LIN {X 0.029,Y -586.530,Z 530.477,A 0.000,B 0.000,C 90.000,E1 301.799} C_DIS
LIN {X 0.083,Y -590.989,Z 530.474,A 0.000,B 0.000,C 90.000,E1 301.258} C_DIS
LIN {X 0.018,Y -595.734,Z 530.471,A 0.000,B 0.000,C 90.000,E1 300.747} C_DIS
LIN {X 0.138,Y -599.927,Z 530.468,A 0.000,B 0.000,C 90.000,E1 300.207} C_DIS
LIN {X 0.251,Y -604.747,Z 530.464,A 0.000,B 0.000,C 90.000,E1 299.539} C_DIS
LIN {X 0.334,Y -611.596,Z 530.458,A 0.000,B 0.000,C 90.000,E1 298.487} C_DIS
LIN {X 0.265,Y -614.592,Z 530.456,A 0.000,B 0.000,C 90.000,E1 297.975} C_DIS
LIN {X 0.227,Y -616.501,Z 530.453,A 0.000,B 0.000,C 90.000,E1 297.590} C_DIS
LIN {X 0.209,Y -617.579,Z 530.452,A 0.000,B 0.000,C 90.000,E1 297.334} C_DIS
LIN {X 0.179,Y -619.100,Z 530.449,A 0.000,B 0.000,C 90.000,E1 296.821} C_DIS
LIN {X 0.170,Y -619.570,Z 530.448,A 0.000,B 0.000,C 90.000,E1 296.565} C_DIS
LIN {X 0.162,Y -619.896,Z 530.446,A 0.000,B 0.000,C 90.000,E1 296.309} C_DIS
LIN {X 0.157,Y -620.039,Z 530.445,A 0.000,B 0.000,C 90.000,E1 296.052} C_DIS
LIN {X 0.146,Y -619.660,Z 530.442,A 0.000,B 0.000,C 90.000,E1 295.540} C_DIS
LIN {X 0.140,Y -619.341,Z 530.441,A 0.000,B 0.000,C 90.000,E1 295.283} C_DIS
LIN {X 0.133,Y -618.398,Z 530.439,A 0.000,B 0.000,C 90.000,E1 295.027} C_DIS
LIN {X 0.123,Y -617.735,Z 530.438,A 0.000,B 0.000,C 90.000,E1 294.771} C_DIS
LIN {X 0.117,Y -617.127,Z 530.437,A 0.000,B 0.000,C 90.000,E1 294.643} C_DIS
LIN {X 0.110,Y -616.003,Z 530.436,A 0.000,B 0.000,C 90.000,E1 294.515} C_DIS
LIN {X 0.101,Y -615.099,Z 530.436,A 0.000,B 0.000,C 90.000,E1 294.387} C_DIS
LIN {X 0.079,Y -613.630,Z 530.434,A 0.000,B 0.000,C 90.000,E1 294.131} C_DIS
LIN {X -0.183,Y -612.297,Z 530.433,A 0.000,B 0.000,C 90.000,E1 294.027} C_DIS
LIN {X -0.142,Y -610.741,Z 530.433,A 0.000,B 0.000,C 90.000,E1 293.898} C_DIS
LIN {X -0.099,Y -607.183,Z 530.431,A 0.000,B 0.000,C 90.000,E1 293.567} C_DIS
LIN {X -0.081,Y -600.309,Z 530.429,A 0.000,B 0.000,C 90.000,E1 293.131} C_DIS
LIN {X 0.139,Y -594.236,Z 530.427,A 0.000,B 0.000,C 90.000,E1 292.845} C_DIS
LIN {X -0.178,Y -586.014,Z 530.425,A 0.000,B 0.000,C 90.000,E1 292.514} C_DIS
LIN {X 0.007,Y -580.558,Z 530.423,A 0.000,B 0.000,C 90.000,E1 292.206} C_DIS
LIN {X -0.138,Y -578.106,Z 530.422,A 0.000,B 0.000,C 90.000,E1 292.025} C_DIS
LIN {X -0.120,Y -576.577,Z 530.421,A 0.000,B 0.000,C 90.000,E1 291.844} C_DIS
LIN {X -0.128,Y -575.849,Z 530.420,A 0.000,B 0.000,C 90.000,E1 291.642} C_DIS
LIN {X 0.113,Y -575.619,Z 530.419,A 0.000,B 0.000,C 90.000,E1 291.461} C_DIS
LIN {X -0.080,Y -575.495,Z 530.414,A 0.000,B 0.000,C 90.000,E1 290.482} C_DIS
LIN {X 0.294,Y -575.816,Z 530.409,A 0.000,B 0.000,C 90.000,E1 289.631} C_DIS
LIN {X -0.234,Y -575.885,Z 530.403,A 0.000,B 0.000,C 90.000,E1 288.598} C_DIS
LIN {X -0.026,Y -575.856,Z 530.396,A 0.000,B 0.000,C 90.000,E1 287.221} C_DIS
LIN {X 0.184,Y -575.564,Z 530.388,A 0.000,B 0.000,C 90.000,E1 285.843} C_DIS
LIN {X 0.081,Y -574.849,Z 530.378,A 0.000,B 0.000,C 90.000,E1 283.953} C_DIS
LIN {X 0.114,Y -574.340,Z 530.370,A 0.000,B 0.000,C 90.000,E1 282.591} C_DIS
LIN {X 0.204,Y -573.645,Z 530.361,A 0.000,B 0.000,C 90.000,E1 280.950} C_DIS
LIN {X 0.169,Y -572.922,Z 530.352,A 0.000,B 0.000,C 90.000,E1 279.321} C_DIS
LIN {X -0.235,Y -572.026,Z 530.340,A 0.000,B 0.000,C 90.000,E1 277.182} C_DIS
LIN {X -0.193,Y -571.609,Z 530.334,A 0.000,B 0.000,C 90.000,E1 276.087} C_DIS
LIN {X 0.016,Y -571.061,Z 530.326,A 0.000,B 0.000,C 90.000,E1 274.702} C_DIS
LIN {X 0.120,Y -570.353,Z 530.319,A 0.000,B 0.000,C 90.000,E1 273.326} C_DIS
LIN {X 0.094,Y -569.713,Z 530.313,A 0.000,B 0.000,C 90.000,E1 272.236} C_DIS
LIN {X 0.179,Y -568.765,Z 530.305,A 0.000,B 0.000,C 90.000,E1 270.859} C_DIS
LIN {X 0.111,Y -567.916,Z 530.299,A 0.000,B 0.000,C 90.000,E1 269.771} C_DIS
LIN {X -0.167,Y -566.298,Z 530.288,A 0.000,B 0.000,C 90.000,E1 267.879} C_DIS
LIN {X -0.032,Y -564.887,Z 530.279,A 0.000,B 0.000,C 90.000,E1 266.216} C_DIS
LIN {X 0.000,Y -563.746,Z 530.271,A 0.000,B 0.000,C 90.000,E1 264.837} C_DIS
LIN {X 0.072,Y -562.379,Z 530.264,A 0.000,B 0.000,C 90.000,E1 263.451} C_DIS
LIN {X -0.024,Y -561.272,Z 530.258,A 0.000,B 0.000,C 90.000,E1 262.356} C_DIS
LIN {X -0.002,Y -559.763,Z 530.250,A 0.000,B 0.000,C 90.000,E1 260.971} C_DIS
LIN {X 0.212,Y -557.715,Z 530.241,A 0.000,B 0.000,C 90.000,E1 259.285} C_DIS
LIN {X -0.058,Y -555.607,Z 530.231,A 0.000,B 0.000,C 90.000,E1 257.645} C_DIS
LIN {X 0.046,Y -554.014,Z 530.225,A 0.000,B 0.000,C 90.000,E1 256.520} C_DIS
LIN {X 0.113,Y -551.877,Z 530.217,A 0.000,B 0.000,C 90.000,E1 255.117} C_DIS
LIN {X -0.117,Y -549.518,Z 530.210,A 0.000,B 0.000,C 90.000,E1 253.740} C_DIS
LIN {X -0.196,Y -548.025,Z 530.205,A 0.000,B 0.000,C 90.000,E1 252.906} C_DIS
LIN {X 0.199,Y -545.202,Z 530.197,A 0.000,B 0.000,C 90.000,E1 251.456} C_DIS
LIN {X -0.211,Y -542.867,Z 530.191,A 0.000,B 0.000,C 90.000,E1 250.369} C_DIS
LIN {X 0.039,Y -540.458,Z 530.185,A 0.000,B 0.000,C 90.000,E1 249.209} C_DIS
LIN {X -0.252,Y -537.864,Z 530.178,A 0.000,B 0.000,C 90.000,E1 248.103} C_DIS
LIN {X 0.119,Y -535.177,Z 530.172,A 0.000,B 0.000,C 90.000,E1 246.922} C_DIS
LIN {X -0.040,Y -532.319,Z 530.166,A 0.000,B 0.000,C 90.000,E1 245.793} C_DIS
LIN {X -0.240,Y -529.288,Z 530.159,A 0.000,B 0.000,C 90.000,E1 244.665} C_DIS
LIN {X -0.092,Y -525.356,Z 530.151,A 0.000,B 0.000,C 90.000,E1 243.204} C_DIS
LIN {X 0.140,Y -520.454,Z 530.141,A 0.000,B 0.000,C 90.000,E1 241.435} C_DIS
LIN {X -0.096,Y -516.317,Z 530.133,A 0.000,B 0.000,C 90.000,E1 239.999} C_DIS
LIN {X -0.157,Y -513.781,Z 530.128,A 0.000,B 0.000,C 90.000,E1 239.125} C_DIS
LIN {X 0.075,Y -508.474,Z 530.119,A 0.000,B 0.000,C 90.000,E1 237.327} C_DIS
LIN {X 0.100,Y -504.834,Z 530.112,A 0.000,B 0.000,C 90.000,E1 236.135} C_DIS
LIN {X 0.283,Y -496.859,Z 530.097,A 0.000,B 0.000,C 90.000,E1 233.417} C_DIS
LIN {X 0.143,Y -491.747,Z 530.087,A 0.000,B 0.000,C 90.000,E1 231.618} C_DIS
LIN {X -0.039,Y -485.884,Z 530.075,A 0.000,B 0.000,C 90.000,E1 229.504} C_DIS
LIN {X 0.314,Y -480.233,Z 530.063,A 0.000,B 0.000,C 90.000,E1 227.310} C_DIS
LIN {X 0.128,Y -474.745,Z 530.051,A 0.000,B 0.000,C 90.000,E1 225.162} C_DIS
LIN {X 0.041,Y -470.153,Z 530.041,A 0.000,B 0.000,C 90.000,E1 223.299} C_DIS
LIN {X -0.203,Y -466.470,Z 530.032,A 0.000,B 0.000,C 90.000,E1 221.757} C_DIS
LIN {X -0.162,Y -462.896,Z 530.023,A 0.000,B 0.000,C 90.000,E1 220.172} C_DIS
LIN {X -0.071,Y -457.922,Z 530.011,A 0.000,B 0.000,C 90.000,E1 217.935} C_DIS
LIN {X -0.044,Y -453.772,Z 530.000,A 0.000,B 0.000,C 90.000,E1 216.011} C_DIS
LIN {X -0.292,Y -449.120,Z 529.988,A 0.000,B 0.000,C 90.000,E1 213.785} C_DIS
LIN {X 0.017,Y -445.273,Z 529.977,A 0.000,B 0.000,C 90.000,E1 211.799} C_DIS
LIN {X -0.233,Y -441.608,Z 529.966,A 0.000,B 0.000,C 90.000,E1 209.873} C_DIS
LIN {X 0.062,Y -436.926,Z 529.951,A 0.000,B 0.000,C 90.000,E1 207.206} C_DIS
LIN {X 0.174,Y -433.585,Z 529.940,A 0.000,B 0.000,C 90.000,E1 205.207} C_DIS
LIN {X -0.151,Y -429.254,Z 529.925,A 0.000,B 0.000,C 90.000,E1 202.589} C_DIS
LIN {X 0.038,Y -426.248,Z 529.914,A 0.000,B 0.000,C 90.000,E1 200.556} C_DIS
LIN {X -0.027,Y -422.603,Z 529.899,A 0.000,B 0.000,C 90.000,E1 197.873} C_DIS
LIN {X -0.014,Y -420.158,Z 529.888,A 0.000,B 0.000,C 90.000,E1 195.843} C_DIS
LIN {X -0.170,Y -417.666,Z 529.877,A 0.000,B 0.000,C 90.000,E1 193.828} C_DIS
LIN {X 0.017,Y -414.393,Z 529.862,A 0.000,B 0.000,C 90.000,E1 191.074} C_DIS
LIN {X -0.060,Y -412.170,Z 529.850,A 0.000,B 0.000,C 90.000,E1 189.029} C_DIS
LIN {X 0.076,Y -409.962,Z 529.839,A 0.000,B 0.000,C 90.000,E1 186.947} C_DIS
LIN {X 0.083,Y -407.486,Z 529.825,A 0.000,B 0.000,C 90.000,E1 184.531} C_DIS
LIN {X -0.068,Y -404.960,Z 529.808,A 0.000,B 0.000,C 90.000,E1 181.432} C_DIS
LIN {X 0.098,Y -403.164,Z 529.792,A 0.000,B 0.000,C 90.000,E1 178.625} C_DIS
LIN {X 0.194,Y -401.751,Z 529.773,A 0.000,B 0.000,C 90.000,E1 175.122} C_DIS
LIN {X -0.034,Y -401.225,Z 529.754,A 0.000,B 0.000,C 90.000,E1 171.659} C_DIS
LIN {X -0.104,Y -401.303,Z 529.736,A 0.000,B 0.000,C 90.000,E1 168.522} C_DIS
LIN {X 0.005,Y -401.663,Z 529.725,A 0.000,B 0.000,C 90.000,E1 166.408} C_DIS
LIN {X -0.086,Y -402.363,Z 529.711,A 0.000,B 0.000,C 90.000,E1 163.976} C_DIS
LIN {X -0.022,Y -403.222,Z 529.699,A 0.000,B 0.000,C 90.000,E1 161.873} C_DIS
LIN {X 0.091,Y -404.081,Z 529.690,A 0.000,B 0.000,C 90.000,E1 160.115} C_DIS
LIN {X 0.085,Y -405.290,Z 529.678,A 0.000,B 0.000,C 90.000,E1 158.028} C_DIS
LIN {X -0.007,Y -406.392,Z 529.668,A 0.000,B 0.000,C 90.000,E1 156.305} C_DIS
LIN {X -0.028,Y -407.892,Z 529.657,A 0.000,B 0.000,C 90.000,E1 154.229} C_DIS
LIN {X -0.211,Y -408.880,Z 529.649,A 0.000,B 0.000,C 90.000,E1 152.871} C_DIS
LIN {X -0.095,Y -410.059,Z 529.640,A 0.000,B 0.000,C 90.000,E1 151.129} C_DIS
LIN {X -0.119,Y -411.164,Z 529.630,A 0.000,B 0.000,C 90.000,E1 149.410} C_DIS
LIN {X 0.089,Y -412.047,Z 529.620,A 0.000,B 0.000,C 90.000,E1 147.661} C_DIS
LIN {X 0.036,Y -412.707,Z 529.613,A 0.000,B 0.000,C 90.000,E1 146.294} C_DIS
LIN {X 0.154,Y -413.430,Z 529.603,A 0.000,B 0.000,C 90.000,E1 144.562} C_DIS
LIN {X 0.015,Y -413.913,Z 529.596,A 0.000,B 0.000,C 90.000,E1 143.210} C_DIS
LIN {X 0.138,Y -414.317,Z 529.588,A 0.000,B 0.000,C 90.000,E1 141.823} C_DIS
LIN {X -0.138,Y -414.733,Z 529.579,A 0.000,B 0.000,C 90.000,E1 140.150} C_DIS
LIN {X 0.121,Y -415.020,Z 529.569,A 0.000,B 0.000,C 90.000,E1 138.405} C_DIS
LIN {X 0.075,Y -415.151,Z 529.560,A 0.000,B 0.000,C 90.000,E1 136.701} C_DIS
LIN {X 0.019,Y -415.283,Z 529.550,A 0.000,B 0.000,C 90.000,E1 135.000} C_DIS
LIN {X 0.094,Y -415.259,Z 529.542,A 0.000,B 0.000,C 90.000,E1 133.623} C_DIS
LIN {X -0.122,Y -415.113,Z 529.535,A 0.000,B 0.000,C 90.000,E1 132.285} C_DIS
LIN {X 0.100,Y -414.856,Z 529.529,A 0.000,B 0.000,C 90.000,E1 131.229} C_DIS
LIN {X 0.006,Y -414.525,Z 529.523,A 0.000,B 0.000,C 90.000,E1 130.216} C_DIS
LIN {X 0.132,Y -413.810,Z 529.516,A 0.000,B 0.000,C 90.000,E1 128.830} C_DIS
LIN {X -0.100,Y -412.607,Z 529.505,A 0.000,B 0.000,C 90.000,E1 126.950} C_DIS
LIN {X -0.139,Y -412.622,Z 529.505,A 0.000,B 0.000,C 90.000,E1 126.950} C_DIS
LIN {X 0.107,Y -415.118,Z 529.501,A 0.000,B 0.000,C 90.000,E1 126.091} C_DIS
LIN {X 0.038,Y -416.033,Z 529.499,A 0.000,B 0.000,C 90.000,E1 125.758} C_DIS
LIN {X 0.167,Y -425.545,Z 529.478,A 0.000,B 0.000,C 90.000,E1 122.005} C_DIS
LIN {X 0.111,Y -430.577,Z 529.469,A 0.000,B 0.000,C 90.000,E1 120.335} C_DIS
LIN {X -0.088,Y -441.486,Z 529.445,A 0.000,B 0.000,C 90.000,E1 116.052} C_DIS
LIN {X -0.170,Y -444.400,Z 529.439,A 0.000,B 0.000,C 90.000,E1 115.079} C_DIS
LIN {X 0.089,Y -445.210,Z 529.437,A 0.000,B 0.000,C 90.000,E1 114.719} C_DIS
LIN {X -0.211,Y -450.645,Z 529.424,A 0.000,B 0.000,C 90.000,E1 112.333} C_DIS
LIN {X 0.167,Y -450.745,Z 529.424,A 0.000,B 0.000,C 90.000,E1 112.280} C_DIS
LIN {X 0.034,Y -472.851,Z 529.419,A 0.000,B 0.000,C 90.000,E1 111.461} C_DIS
LIN {X 0.234,Y -486.897,Z 529.416,A 0.000,B 0.000,C 90.000,E1 110.918} C_DIS
LIN {X -0.093,Y -497.259,Z 529.414,A 0.000,B 0.000,C 90.000,E1 110.556} C_DIS
LIN {X 0.107,Y -507.656,Z 529.412,A 0.000,B 0.000,C 90.000,E1 110.120} C_DIS
LIN {X 0.088,Y -524.687,Z 529.408,A 0.000,B 0.000,C 90.000,E1 109.396} C_DIS
LIN {X 0.158,Y -531.308,Z 529.406,A 0.000,B 0.000,C 90.000,E1 109.087} C_DIS
LIN {X -0.203,Y -539.551,Z 529.404,A 0.000,B 0.000,C 90.000,E1 108.725} C_DIS
LIN {X -0.070,Y -547.732,Z 529.402,A 0.000,B 0.000,C 90.000,E1 108.290} C_DIS
LIN {X -0.110,Y -553.800,Z 529.400,A 0.000,B 0.000,C 90.000,E1 107.928} C_DIS
LIN {X 0.065,Y -559.931,Z 529.397,A 0.000,B 0.000,C 90.000,E1 107.511} C_DIS
LIN {X -0.211,Y -564.414,Z 529.396,A 0.000,B 0.000,C 90.000,E1 107.221} C_DIS
LIN {X 0.119,Y -570.062,Z 529.393,A 0.000,B 0.000,C 90.000,E1 106.732} C_DIS
LIN {X -0.311,Y -576.431,Z 529.390,A 0.000,B 0.000,C 90.000,E1 106.205} C_DIS
LIN {X -0.004,Y -581.131,Z 529.387,A 0.000,B 0.000,C 90.000,E1 105.717} C_DIS
LIN {X 0.197,Y -585.870,Z 529.385,A 0.000,B 0.000,C 90.000,E1 105.190} C_DIS
LIN {X 0.043,Y -591.085,Z 529.381,A 0.000,B 0.000,C 90.000,E1 104.592} C_DIS
LIN {X 0.077,Y -594.163,Z 529.379,A 0.000,B 0.000,C 90.000,E1 104.189} C_DIS
LIN {X 0.204,Y -596.933,Z 529.377,A 0.000,B 0.000,C 90.000,E1 103.828} C_DIS
LIN {X -0.180,Y -601.596,Z 529.373,A 0.000,B 0.000,C 90.000,E1 103.231} C_DIS
LIN {X 0.166,Y -607.111,Z 529.369,A 0.000,B 0.000,C 90.000,E1 102.411} C_DIS
LIN {X -0.146,Y -612.403,Z 529.365,A 0.000,B 0.000,C 90.000,E1 101.658} C_DIS
LIN {X 0.143,Y -614.897,Z 529.363,A 0.000,B 0.000,C 90.000,E1 101.243} C_DIS
LIN {X 0.087,Y -618.731,Z 529.359,A 0.000,B 0.000,C 90.000,E1 100.602} C_DIS
LIN {X -0.112,Y -623.582,Z 529.354,A 0.000,B 0.000,C 90.000,E1 99.726} C_DIS
LIN {X 0.150,Y -628.784,Z 529.348,A 0.000,B 0.000,C 90.000,E1 98.681} C_DIS
LIN {X -0.088,Y -632.983,Z 529.343,A 0.000,B 0.000,C 90.000,E1 97.814} C_DIS
LIN {X -0.056,Y -638.719,Z 529.336,A 0.000,B 0.000,C 90.000,E1 96.549} C_DIS
LIN {X -0.310,Y -643.120,Z 529.331,A 0.000,B 0.000,C 90.000,E1 95.568} C_DIS
LIN {X 0.130,Y -647.072,Z 529.325,A 0.000,B 0.000,C 90.000,E1 94.531} C_DIS
LIN {X -0.280,Y -648.842,Z 529.323,A 0.000,B 0.000,C 90.000,E1 94.069} C_DIS
LIN {X 0.180,Y -651.969,Z 529.317,A 0.000,B 0.000,C 90.000,E1 93.037} C_DIS
LIN {X 0.208,Y -653.937,Z 529.313,A 0.000,B 0.000,C 90.000,E1 92.293} C_DIS
LIN {X -0.193,Y -655.062,Z 529.310,A 0.000,B 0.000,C 90.000,E1 91.835} C_DIS
LIN {X 0.086,Y -655.977,Z 529.307,A 0.000,B 0.000,C 90.000,E1 91.318} C_DIS
LIN {X 0.161,Y -656.981,Z 529.303,A 0.000,B 0.000,C 90.000,E1 90.573} C_DIS
LIN {X 0.249,Y -657.557,Z 529.299,A 0.000,B 0.000,C 90.000,E1 89.828} C_DIS
LIN {X -0.128,Y -657.756,Z 529.297,A 0.000,B 0.000,C 90.000,E1 89.370} C_DIS
LIN {X -0.036,Y -657.710,Z 529.292,A 0.000,B 0.000,C 90.000,E1 88.625} C_DIS
LIN {X 0.263,Y -657.468,Z 529.290,A 0.000,B 0.000,C 90.000,E1 88.108} C_DIS
LIN {X -0.114,Y -657.097,Z 529.287,A 0.000,B 0.000,C 90.000,E1 87.650} C_DIS
LIN {X 0.159,Y -656.594,Z 529.284,A 0.000,B 0.000,C 90.000,E1 87.135} C_DIS
LIN {X 0.264,Y -655.543,Z 529.280,A 0.000,B 0.000,C 90.000,E1 86.388} C_DIS
LIN {X 0.066,Y -655.167,Z 529.279,A 0.000,B 0.000,C 90.000,E1 86.159} C_DIS
LIN {X 0.005,Y -653.002,Z 529.273,A 0.000,B 0.000,C 90.000,E1 85.179} C_DIS
LIN {X 0.233,Y -651.736,Z 529.271,A 0.000,B 0.000,C 90.000,E1 84.666} C_DIS
LIN {X -0.291,Y -649.710,Z 529.266,A 0.000,B 0.000,C 90.000,E1 83.970} C_DIS
LIN {X -0.252,Y -647.309,Z 529.262,A 0.000,B 0.000,C 90.000,E1 83.223} C_DIS
LIN {X -0.005,Y -645.607,Z 529.260,A 0.000,B 0.000,C 90.000,E1 82.704} C_DIS
LIN {X 0.230,Y -643.765,Z 529.257,A 0.000,B 0.000,C 90.000,E1 82.186} C_DIS
LIN {X -0.155,Y -638.588,Z 529.250,A 0.000,B 0.000,C 90.000,E1 80.971} C_DIS
LIN {X -0.047,Y -635.076,Z 529.246,A 0.000,B 0.000,C 90.000,E1 80.208} C_DIS
LIN {X -0.084,Y -631.229,Z 529.241,A 0.000,B 0.000,C 90.000,E1 79.454} C_DIS
LIN {X 0.153,Y -628.532,Z 529.239,A 0.000,B 0.000,C 90.000,E1 78.926} C_DIS
LIN {X 0.041,Y -624.252,Z 529.234,A 0.000,B 0.000,C 90.000,E1 78.173} C_DIS
LIN {X 0.185,Y -620.505,Z 529.231,A 0.000,B 0.000,C 90.000,E1 77.521} C_DIS
LIN {X 0.166,Y -616.560,Z 529.227,A 0.000,B 0.000,C 90.000,E1 76.881} C_DIS
LIN {X -0.110,Y -613.895,Z 529.225,A 0.000,B 0.000,C 90.000,E1 76.520} C_DIS
LIN {X -0.018,Y -609.352,Z 529.222,A 0.000,B 0.000,C 90.000,E1 75.880} C_DIS
LIN {X 0.008,Y -604.041,Z 529.218,A 0.000,B 0.000,C 90.000,E1 75.227} C_DIS
LIN {X -0.008,Y -598.104,Z 529.214,A 0.000,B 0.000,C 90.000,E1 74.574} C_DIS
LIN {X 0.044,Y -593.055,Z 529.211,A 0.000,B 0.000,C 90.000,E1 74.047} C_DIS
LIN {X -0.147,Y -587.757,Z 529.209,A 0.000,B 0.000,C 90.000,E1 73.559} C_DIS
LIN {X -0.169,Y -583.572,Z 529.207,A 0.000,B 0.000,C 90.000,E1 73.196} C_DIS
LIN {X -0.100,Y -577.818,Z 529.204,A 0.000,B 0.000,C 90.000,E1 72.725} C_DIS
LIN {X 0.183,Y -571.779,Z 529.202,A 0.000,B 0.000,C 90.000,E1 72.253} C_DIS
LIN {X 0.113,Y -567.221,Z 529.200,A 0.000,B 0.000,C 90.000,E1 71.945} C_DIS
LIN {X -0.147,Y -560.899,Z 529.198,A 0.000,B 0.000,C 90.000,E1 71.583} C_DIS
LIN {X 0.080,Y -555.796,Z 529.196,A 0.000,B 0.000,C 90.000,E1 71.275} C_DIS
LIN {X 0.292,Y -548.965,Z 529.194,A 0.000,B 0.000,C 90.000,E1 70.913} C_DIS
LIN {X -0.176,Y -543.682,Z 529.193,A 0.000,B 0.000,C 90.000,E1 70.732} C_DIS
LIN {X 0.066,Y -536.315,Z 529.191,A 0.000,B 0.000,C 90.000,E1 70.423} C_DIS
LIN {X -0.028,Y -528.724,Z 529.190,A 0.000,B 0.000,C 90.000,E1 70.188} C_DIS
LIN {X -0.075,Y -517.819,Z 529.188,A 0.000,B 0.000,C 90.000,E1 69.880} C_DIS
LIN {X 0.136,Y -504.950,Z 529.186,A 0.000,B 0.000,C 90.000,E1 69.518} C_DIS
LIN {X 0.022,Y -493.745,Z 529.185,A 0.000,B 0.000,C 90.000,E1 69.263} C_DIS
LIN {X -0.065,Y -468.161,Z 529.182,A 0.000,B 0.000,C 90.000,E1 68.720} C_DIS
LIN {X -0.106,Y -468.029,Z 529.182,A 0.000,B 0.000,C 90.000,E1 68.720} C_DIS
LIN {X -0.010,Y -465.707,Z 529.173,A 0.000,B 0.000,C 90.000,E1 67.102} C_DIS
LIN {X -0.213,Y -456.175,Z 529.146,A 0.000,B 0.000,C 90.000,E1 62.359} C_DIS
LIN {X -0.107,Y -455.659,Z 529.145,A 0.000,B 0.000,C 90.000,E1 62.025} C_DIS
LIN {X -0.116,Y -454.168,Z 529.141,A 0.000,B 0.000,C 90.000,E1 61.385} C_DIS
LIN {X -0.013,Y -445.139,Z 529.118,A 0.000,B 0.000,C 90.000,E1 57.168} C_DIS
LIN {X 0.146,Y -444.719,Z 529.116,A 0.000,B 0.000,C 90.000,E1 56.914} C_DIS
LIN {X 0.107,Y -444.713,Z 529.116,A 0.000,B 0.000,C 90.000,E1 56.914} C_DIS
LIN {X -0.141,Y -447.404,Z 529.110,A 0.000,B 0.000,C 90.000,E1 55.881} C_DIS
LIN {X -0.055,Y -449.804,Z 529.105,A 0.000,B 0.000,C 90.000,E1 54.895} C_DIS
LIN {X 0.137,Y -452.660,Z 529.098,A 0.000,B 0.000,C 90.000,E1 53.577} C_DIS
LIN {X -0.081,Y -454.649,Z 529.092,A 0.000,B 0.000,C 90.000,E1 52.637} C_DIS
LIN {X 0.091,Y -457.039,Z 529.085,A 0.000,B 0.000,C 90.000,E1 51.331} C_DIS
LIN {X -0.058,Y -459.147,Z 529.078,A 0.000,B 0.000,C 90.000,E1 50.070} C_DIS
LIN {X 0.087,Y -460.572,Z 529.073,A 0.000,B 0.000,C 90.000,E1 49.094} C_DIS
LIN {X -0.051,Y -462.327,Z 529.066,A 0.000,B 0.000,C 90.000,E1 47.838} C_DIS
LIN {X 0.127,Y -463.394,Z 529.060,A 0.000,B 0.000,C 90.000,E1 46.863} C_DIS
LIN {X 0.295,Y -464.274,Z 529.055,A 0.000,B 0.000,C 90.000,E1 45.891} C_DIS
LIN {X -0.181,Y -464.979,Z 529.050,A 0.000,B 0.000,C 90.000,E1 45.000} C_DIS
LIN {X 0.009,Y -465.550,Z 529.045,A 0.000,B 0.000,C 90.000,E1 44.028} C_DIS
LIN {X -0.052,Y -466.008,Z 529.038,A 0.000,B 0.000,C 90.000,E1 42.771} C_DIS
LIN {X -0.110,Y -466.200,Z 529.031,A 0.000,B 0.000,C 90.000,E1 41.515} C_DIS
LIN {X -0.123,Y -466.180,Z 529.024,A 0.000,B 0.000,C 90.000,E1 40.253} C_DIS
LIN {X -0.080,Y -465.827,Z 529.015,A 0.000,B 0.000,C 90.000,E1 38.669} C_DIS
LIN {X -0.018,Y -465.413,Z 529.008,A 0.000,B 0.000,C 90.000,E1 37.397} C_DIS
LIN {X -0.052,Y -464.866,Z 529.001,A 0.000,B 0.000,C 90.000,E1 36.137} C_DIS
LIN {X 0.130,Y -464.089,Z 528.992,A 0.000,B 0.000,C 90.000,E1 34.532} C_DIS
LIN {X 0.040,Y -463.271,Z 528.983,A 0.000,B 0.000,C 90.000,E1 32.959} C_DIS
LIN {X 0.065,Y -462.264,Z 528.973,A 0.000,B 0.000,C 90.000,E1 31.052} C_DIS
LIN {X -0.009,Y -461.101,Z 528.962,A 0.000,B 0.000,C 90.000,E1 29.155} C_DIS
LIN {X -0.012,Y -460.156,Z 528.953,A 0.000,B 0.000,C 90.000,E1 27.564} C_DIS
LIN {X -0.039,Y -458.860,Z 528.941,A 0.000,B 0.000,C 90.000,E1 25.335} C_DIS
LIN {X -0.051,Y -457.482,Z 528.925,A 0.000,B 0.000,C 90.000,E1 22.461} C_DIS
LIN {X 0.071,Y -456.516,Z 528.911,A 0.000,B 0.000,C 90.000,E1 19.885} C_DIS
LIN {X -0.231,Y -455.958,Z 528.900,A 0.000,B 0.000,C 90.000,E1 18.000} C_DIS
LIN {X 0.069,Y -455.540,Z 528.887,A 0.000,B 0.000,C 90.000,E1 15.717} C_DIS
LIN {X -0.128,Y -455.496,Z 528.873,A 0.000,B 0.000,C 90.000,E1 13.175} C_DIS
LIN {X -0.071,Y -455.741,Z 528.862,A 0.000,B 0.000,C 90.000,E1 11.243} C_DIS
LIN {X 0.134,Y -456.142,Z 528.854,A 0.000,B 0.000,C 90.000,E1 9.613} C_DIS
LIN {X -0.180,Y -456.977,Z 528.841,A 0.000,B 0.000,C 90.000,E1 7.409} C_DIS
LIN {X -0.188,Y -458.469,Z 528.825,A 0.000,B 0.000,C 90.000,E1 4.531} C_DIS
LIN {X -0.213,Y -460.480,Z 528.809,A 0.000,B 0.000,C 90.000,E1 1.661} C_DIS
LIN {X 0.092,Y -463.469,Z 528.792,A 0.000,B 0.000,C 90.000,E1 358.511} C_DIS
LIN {X 0.009,Y -466.426,Z 528.778,A 0.000,B 0.000,C 90.000,E1 355.988} C_DIS
LIN {X -0.140,Y -469.266,Z 528.766,A 0.000,B 0.000,C 90.000,E1 353.799} C_DIS
LIN {X 0.030,Y -471.824,Z 528.755,A 0.000,B 0.000,C 90.000,E1 351.894} C_DIS
LIN {X -0.147,Y -474.456,Z 528.745,A 0.000,B 0.000,C 90.000,E1 350.038} C_DIS
LIN {X 0.124,Y -477.613,Z 528.732,A 0.000,B 0.000,C 90.000,E1 347.825} C_DIS
LIN {X 0.049,Y -482.343,Z 528.717,A 0.000,B 0.000,C 90.000,E1 345.046} C_DIS
LIN {X -0.062,Y -487.141,Z 528.703,A 0.000,B 0.000,C 90.000,E1 342.598} C_DIS
LIN {X 0.240,Y -491.377,Z 528.691,A 0.000,B 0.000,C 90.000,E1 340.423} C_DIS
LIN {X -0.200,Y -494.446,Z 528.683,A 0.000,B 0.000,C 90.000,E1 338.954} C_DIS
LIN {X 0.056,Y -497.484,Z 528.675,A 0.000,B 0.000,C 90.000,E1 337.411} C_DIS
LIN {X -0.094,Y -500.438,Z 528.666,A 0.000,B 0.000,C 90.000,E1 335.921} C_DIS
LIN {X 0.009,Y -503.294,Z 528.658,A 0.000,B 0.000,C 90.000,E1 334.409} C_DIS
LIN {X 0.079,Y -505.543,Z 528.651,A 0.000,B 0.000,C 90.000,E1 333.204} C_DIS
LIN {X -0.082,Y -508.891,Z 528.641,A 0.000,B 0.000,C 90.000,E1 331.435} C_DIS
LIN {X -0.060,Y -511.608,Z 528.633,A 0.000,B 0.000,C 90.000,E1 329.950} C_DIS
LIN {X 0.083,Y -515.525,Z 528.622,A 0.000,B 0.000,C 90.000,E1 327.867} C_DIS
LIN {X 0.176,Y -519.503,Z 528.610,A 0.000,B 0.000,C 90.000,E1 325.801} C_DIS
LIN {X -0.014,Y -522.891,Z 528.600,A 0.000,B 0.000,C 90.000,E1 324.069} C_DIS
LIN {X 0.004,Y -527.381,Z 528.588,A 0.000,B 0.000,C 90.000,E1 321.743} C_DIS
LIN {X 0.169,Y -531.313,Z 528.576,A 0.000,B 0.000,C 90.000,E1 319.703} C_DIS
LIN {X -0.031,Y -534.844,Z 528.567,A 0.000,B 0.000,C 90.000,E1 318.000} C_DIS
LIN {X 0.248,Y -537.864,Z 528.559,A 0.000,B 0.000,C 90.000,E1 316.539} C_DIS
LIN {X 0.175,Y -541.433,Z 528.549,A 0.000,B 0.000,C 90.000,E1 314.838} C_DIS
LIN {X 0.198,Y -545.781,Z 528.538,A 0.000,B 0.000,C 90.000,E1 312.852} C_DIS
LIN {X -0.002,Y -551.025,Z 528.526,A 0.000,B 0.000,C 90.000,E1 310.620} C_DIS
LIN {X 0.158,Y -553.510,Z 528.519,A 0.000,B 0.000,C 90.000,E1 309.483} C_DIS
LIN {X 0.073,Y -556.430,Z 528.512,A 0.000,B 0.000,C 90.000,E1 308.096} C_DIS
LIN {X -0.025,Y -561.095,Z 528.499,A 0.000,B 0.000,C 90.000,E1 305.884} C_DIS
LIN {X 0.266,Y -563.347,Z 528.495,A 0.000,B 0.000,C 90.000,E1 305.025} C_DIS
LIN {X 0.235,Y -565.025,Z 528.492,A 0.000,B 0.000,C 90.000,E1 304.532} C_DIS
LIN {X 0.072,Y -565.937,Z 528.491,A 0.000,B 0.000,C 90.000,E1 304.405} C_DIS
LIN {X -0.032,Y -566.650,Z 528.490,A 0.000,B 0.000,C 90.000,E1 304.278} C_DIS
LIN {X -0.020,Y -568.440,Z 528.488,A 0.000,B 0.000,C 90.000,E1 303.865} C_DIS
LIN {X -0.263,Y -573.007,Z 528.484,A 0.000,B 0.000,C 90.000,E1 303.166} C_DIS
LIN {X 0.005,Y -576.942,Z 528.481,A 0.000,B 0.000,C 90.000,E1 302.594} C_DIS
LIN {X -0.162,Y -578.732,Z 528.480,A 0.000,B 0.000,C 90.000,E1 302.339} C_DIS
LIN {X 0.127,Y -590.707,Z 528.471,A 0.000,B 0.000,C 90.000,E1 300.797} C_DIS
LIN {X 0.209,Y -595.150,Z 528.468,A 0.000,B 0.000,C 90.000,E1 300.256} C_DIS
LIN {X 0.067,Y -598.276,Z 528.466,A 0.000,B 0.000,C 90.000,E1 299.873} C_DIS
LIN {X 0.091,Y -604.355,Z 528.461,A 0.000,B 0.000,C 90.000,E1 298.949} C_DIS
LIN {X 0.210,Y -609.242,Z 528.457,A 0.000,B 0.000,C 90.000,E1 298.153} C_DIS
LIN {X 0.144,Y -611.400,Z 528.454,A 0.000,B 0.000,C 90.000,E1 297.769} C_DIS
LIN {X 0.089,Y -613.090,Z 528.452,A 0.000,B 0.000,C 90.000,E1 297.385} C_DIS
LIN {X 0.057,Y -614.127,Z 528.451,A 0.000,B 0.000,C 90.000,E1 297.129} C_DIS
LIN {X 0.027,Y -615.023,Z 528.449,A 0.000,B 0.000,C 90.000,E1 296.873} C_DIS
LIN {X -0.021,Y -615.880,Z 528.446,A 0.000,B 0.000,C 90.000,E1 296.360} C_DIS
LIN {X -0.042,Y -616.087,Z 528.445,A 0.000,B 0.000,C 90.000,E1 296.104} C_DIS
LIN {X -0.081,Y -616.151,Z 528.442,A 0.000,B 0.000,C 90.000,E1 295.591} C_DIS
LIN {X -0.101,Y -615.736,Z 528.441,A 0.000,B 0.000,C 90.000,E1 295.335} C_DIS
LIN {X -0.120,Y -615.134,Z 528.439,A 0.000,B 0.000,C 90.000,E1 295.079} C_DIS
LIN {X -0.143,Y -614.346,Z 528.438,A 0.000,B 0.000,C 90.000,E1 294.823} C_DIS
LIN {X 0.108,Y -611.673,Z 528.435,A 0.000,B 0.000,C 90.000,E1 294.283} C_DIS
LIN {X 0.092,Y -610.646,Z 528.434,A 0.000,B 0.000,C 90.000,E1 294.155} C_DIS
LIN {X 0.221,Y -605.296,Z 528.432,A 0.000,B 0.000,C 90.000,E1 293.643} C_DIS
LIN {X 0.089,Y -600.398,Z 528.430,A 0.000,B 0.000,C 90.000,E1 293.334} C_DIS
LIN {X 0.109,Y -597.505,Z 528.429,A 0.000,B 0.000,C 90.000,E1 293.153} C_DIS
LIN {X 0.229,Y -593.009,Z 528.428,A 0.000,B 0.000,C 90.000,E1 292.950} C_DIS
LIN {X -0.100,Y -587.762,Z 528.426,A 0.000,B 0.000,C 90.000,E1 292.695} C_DIS
LIN {X 0.076,Y -585.714,Z 528.426,A 0.000,B 0.000,C 90.000,E1 292.589} C_DIS
LIN {X 0.202,Y -582.456,Z 528.424,A 0.000,B 0.000,C 90.000,E1 292.386} C_DIS
LIN {X 0.156,Y -579.916,Z 528.424,A 0.000,B 0.000,C 90.000,E1 292.206} C_DIS
LIN {X 0.105,Y -578.603,Z 528.423,A 0.000,B 0.000,C 90.000,E1 292.099} C_DIS
LIN {X -0.264,Y -577.655,Z 528.422,A 0.000,B 0.000,C 90.000,E1 292.025} C_DIS
LIN {X 0.173,Y -576.961,Z 528.421,A 0.000,B 0.000,C 90.000,E1 291.791} C_DIS
LIN {X 0.018,Y -576.457,Z 528.420,A 0.000,B 0.000,C 90.000,E1 291.535} C_DIS
LIN {X -0.215,Y -576.383,Z 528.414,A 0.000,B 0.000,C 90.000,E1 290.610} C_DIS
LIN {X 0.171,Y -576.728,Z 528.410,A 0.000,B 0.000,C 90.000,E1 289.758} C_DIS
LIN {X 0.030,Y -576.829,Z 528.402,A 0.000,B 0.000,C 90.000,E1 288.417} C_DIS
LIN {X 0.255,Y -576.811,Z 528.395,A 0.000,B 0.000,C 90.000,E1 287.040} C_DIS
LIN {X -0.075,Y -576.488,Z 528.387,A 0.000,B 0.000,C 90.000,E1 285.717} C_DIS
LIN {X 0.191,Y -575.928,Z 528.378,A 0.000,B 0.000,C 90.000,E1 284.064} C_DIS
LIN {X 0.111,Y -575.484,Z 528.371,A 0.000,B 0.000,C 90.000,E1 282.715} C_DIS
LIN {X 0.234,Y -574.810,Z 528.362,A 0.000,B 0.000,C 90.000,E1 281.074} C_DIS
LIN {X 0.233,Y -574.123,Z 528.353,A 0.000,B 0.000,C 90.000,E1 279.443} C_DIS
LIN {X -0.244,Y -573.349,Z 528.342,A 0.000,B 0.000,C 90.000,E1 277.587} C_DIS
LIN {X -0.118,Y -572.988,Z 528.336,A 0.000,B 0.000,C 90.000,E1 276.486} C_DIS
LIN {X 0.188,Y -572.303,Z 528.327,A 0.000,B 0.000,C 90.000,E1 274.821} C_DIS
LIN {X -0.211,Y -571.608,Z 528.319,A 0.000,B 0.000,C 90.000,E1 273.498} C_DIS
LIN {X -0.089,Y -570.727,Z 528.312,A 0.000,B 0.000,C 90.000,E1 272.121} C_DIS
LIN {X 0.015,Y -569.763,Z 528.304,A 0.000,B 0.000,C 90.000,E1 270.745} C_DIS
LIN {X 0.088,Y -568.628,Z 528.297,A 0.000,B 0.000,C 90.000,E1 269.370} C_DIS
LIN {X -0.175,Y -566.984,Z 528.286,A 0.000,B 0.000,C 90.000,E1 267.478} C_DIS
LIN {X 0.113,Y -565.272,Z 528.275,A 0.000,B 0.000,C 90.000,E1 265.527} C_DIS
LIN {X 0.055,Y -564.222,Z 528.269,A 0.000,B 0.000,C 90.000,E1 264.432} C_DIS
LIN {X -0.013,Y -563.100,Z 528.263,A 0.000,B 0.000,C 90.000,E1 263.337} C_DIS
LIN {X 0.049,Y -561.585,Z 528.255,A 0.000,B 0.000,C 90.000,E1 261.951} C_DIS
LIN {X 0.015,Y -560.332,Z 528.249,A 0.000,B 0.000,C 90.000,E1 260.849} C_DIS
LIN {X -0.152,Y -557.909,Z 528.238,A 0.000,B 0.000,C 90.000,E1 258.926} C_DIS
LIN {X 0.004,Y -556.121,Z 528.231,A 0.000,B 0.000,C 90.000,E1 257.521} C_DIS
LIN {X -0.008,Y -554.501,Z 528.225,A 0.000,B 0.000,C 90.000,E1 256.408} C_DIS
LIN {X 0.202,Y -552.334,Z 528.217,A 0.000,B 0.000,C 90.000,E1 254.991} C_DIS
LIN {X -0.014,Y -549.907,Z 528.209,A 0.000,B 0.000,C 90.000,E1 253.614} C_DIS
LIN {X -0.087,Y -548.342,Z 528.204,A 0.000,B 0.000,C 90.000,E1 252.779} C_DIS
LIN {X -0.126,Y -544.915,Z 528.195,A 0.000,B 0.000,C 90.000,E1 251.094} C_DIS
LIN {X 0.156,Y -542.510,Z 528.189,A 0.000,B 0.000,C 90.000,E1 249.934} C_DIS
LIN {X -0.102,Y -539.998,Z 528.182,A 0.000,B 0.000,C 90.000,E1 248.827} C_DIS
LIN {X 0.104,Y -537.341,Z 528.176,A 0.000,B 0.000,C 90.000,E1 247.667} C_DIS
LIN {X -0.023,Y -534.556,Z 528.170,A 0.000,B 0.000,C 90.000,E1 246.538} C_DIS
LIN {X 0.101,Y -532.359,Z 528.165,A 0.000,B 0.000,C 90.000,E1 245.665} C_DIS
LIN {X -0.099,Y -529.306,Z 528.159,A 0.000,B 0.000,C 90.000,E1 244.537} C_DIS
LIN {X 0.047,Y -525.306,Z 528.151,A 0.000,B 0.000,C 90.000,E1 243.076} C_DIS
LIN {X 0.277,Y -520.406,Z 528.141,A 0.000,B 0.000,C 90.000,E1 241.307} C_DIS
LIN {X 0.037,Y -516.226,Z 528.133,A 0.000,B 0.000,C 90.000,E1 239.871} C_DIS
LIN {X -0.025,Y -513.663,Z 528.128,A 0.000,B 0.000,C 90.000,E1 238.997} C_DIS
LIN {X -0.135,Y -509.220,Z 528.120,A 0.000,B 0.000,C 90.000,E1 237.533} C_DIS
LIN {X -0.099,Y -505.577,Z 528.113,A 0.000,B 0.000,C 90.000,E1 236.342} C_DIS
LIN {X 0.113,Y -497.501,Z 528.098,A 0.000,B 0.000,C 90.000,E1 233.623} C_DIS
LIN {X -0.154,Y -491.550,Z 528.086,A 0.000,B 0.000,C 90.000,E1 231.537} C_DIS
LIN {X 0.035,Y -485.679,Z 528.074,A 0.000,B 0.000,C 90.000,E1 229.380} C_DIS
LIN {X 0.018,Y -480.040,Z 528.062,A 0.000,B 0.000,C 90.000,E1 227.229} C_DIS
LIN {X -0.170,Y -474.535,Z 528.050,A 0.000,B 0.000,C 90.000,E1 225.081} C_DIS
LIN {X -0.005,Y -470.726,Z 528.042,A 0.000,B 0.000,C 90.000,E1 223.500} C_DIS
LIN {X 0.084,Y -467.000,Z 528.033,A 0.000,B 0.000,C 90.000,E1 221.919} C_DIS
LIN {X 0.185,Y -462.687,Z 528.022,A 0.000,B 0.000,C 90.000,E1 220.011} C_DIS
LIN {X -0.020,Y -457.722,Z 528.010,A 0.000,B 0.000,C 90.000,E1 217.810} C_DIS
LIN {X 0.009,Y -453.578,Z 527.999,A 0.000,B 0.000,C 90.000,E1 215.884} C_DIS
LIN {X 0.010,Y -448.942,Z 527.987,A 0.000,B 0.000,C 90.000,E1 213.627} C_DIS
LIN {X 0.134,Y -444.520,Z 527.974,A 0.000,B 0.000,C 90.000,E1 211.337} C_DIS
LIN {X -0.133,Y -440.849,Z 527.963,A 0.000,B 0.000,C 90.000,E1 209.411} C_DIS
LIN {X -0.107,Y -437.376,Z 527.952,A 0.000,B 0.000,C 90.000,E1 207.436} C_DIS
LIN {X -0.183,Y -434.009,Z 527.941,A 0.000,B 0.000,C 90.000,E1 205.463} C_DIS
LIN {X -0.134,Y -430.155,Z 527.928,A 0.000,B 0.000,C 90.000,E1 203.131} C_DIS
LIN {X 0.068,Y -426.138,Z 527.914,A 0.000,B 0.000,C 90.000,E1 200.429} C_DIS
LIN {X 0.211,Y -422.917,Z 527.901,A 0.000,B 0.000,C 90.000,E1 198.055} C_DIS
LIN {X -0.174,Y -420.438,Z 527.889,A 0.000,B 0.000,C 90.000,E1 196.079} C_DIS
LIN {X 0.082,Y -417.962,Z 527.878,A 0.000,B 0.000,C 90.000,E1 194.008} C_DIS
LIN {X -0.042,Y -414.684,Z 527.863,A 0.000,B 0.000,C 90.000,E1 191.299} C_DIS
LIN {X -0.188,Y -412.466,Z 527.851,A 0.000,B 0.000,C 90.000,E1 189.265} C_DIS
LIN {X -0.068,Y -410.651,Z 527.842,A 0.000,B 0.000,C 90.000,E1 187.530} C_DIS
LIN {X 0.009,Y -408.110,Z 527.828,A 0.000,B 0.000,C 90.000,E1 185.106} C_DIS
LIN {X -0.151,Y -404.933,Z 527.807,A 0.000,B 0.000,C 90.000,E1 181.318} C_DIS
LIN {X 0.015,Y -403.150,Z 527.792,A 0.000,B 0.000,C 90.000,E1 178.511} C_DIS
LIN {X 0.124,Y -401.898,Z 527.774,A 0.000,B 0.000,C 90.000,E1 175.355} C_DIS
LIN {X -0.104,Y -401.332,Z 527.757,A 0.000,B 0.000,C 90.000,E1 172.243} C_DIS
LIN {X -0.152,Y -401.270,Z 527.745,A 0.000,B 0.000,C 90.000,E1 170.151} C_DIS
LIN {X -0.144,Y -401.583,Z 527.730,A 0.000,B 0.000,C 90.000,E1 167.353} C_DIS
LIN {X 0.131,Y -402.294,Z 527.714,A 0.000,B 0.000,C 90.000,E1 164.519} C_DIS
LIN {X -0.224,Y -403.254,Z 527.701,A 0.000,B 0.000,C 90.000,E1 162.127} C_DIS
LIN {X -0.118,Y -404.104,Z 527.691,A 0.000,B 0.000,C 90.000,E1 160.369} C_DIS
LIN {X -0.030,Y -405.548,Z 527.677,A 0.000,B 0.000,C 90.000,E1 157.922} C_DIS
LIN {X -0.073,Y -407.427,Z 527.662,A 0.000,B 0.000,C 90.000,E1 155.153} C_DIS
LIN {X 0.205,Y -408.694,Z 527.652,A 0.000,B 0.000,C 90.000,E1 153.384} C_DIS
LIN {X -0.040,Y -409.915,Z 527.643,A 0.000,B 0.000,C 90.000,E1 151.691} C_DIS
LIN {X 0.094,Y -411.056,Z 527.633,A 0.000,B 0.000,C 90.000,E1 149.950} C_DIS
LIN {X -0.050,Y -412.026,Z 527.624,A 0.000,B 0.000,C 90.000,E1 148.250} C_DIS
LIN {X 0.179,Y -412.918,Z 527.614,A 0.000,B 0.000,C 90.000,E1 146.501} C_DIS
LIN {X -0.106,Y -413.790,Z 527.603,A 0.000,B 0.000,C 90.000,E1 144.482} C_DIS
LIN {X -0.235,Y -414.283,Z 527.595,A 0.000,B 0.000,C 90.000,E1 143.130} C_DIS
LIN {X 0.074,Y -414.785,Z 527.586,A 0.000,B 0.000,C 90.000,E1 141.376} C_DIS
LIN {X 0.074,Y -415.228,Z 527.576,A 0.000,B 0.000,C 90.000,E1 139.666} C_DIS
LIN {X 0.073,Y -415.499,Z 527.567,A 0.000,B 0.000,C 90.000,E1 137.957} C_DIS
LIN {X 0.192,Y -415.686,Z 527.555,A 0.000,B 0.000,C 90.000,E1 135.891} C_DIS
LIN {X -0.021,Y -415.731,Z 527.548,A 0.000,B 0.000,C 90.000,E1 134.555} C_DIS
LIN {X -0.058,Y -415.646,Z 527.538,A 0.000,B 0.000,C 90.000,E1 132.852} C_DIS
LIN {X 0.044,Y -415.367,Z 527.530,A 0.000,B 0.000,C 90.000,E1 131.472} C_DIS
LIN {X 0.138,Y -414.844,Z 527.523,A 0.000,B 0.000,C 90.000,E1 130.092} C_DIS
LIN {X -0.050,Y -414.058,Z 527.515,A 0.000,B 0.000,C 90.000,E1 128.749} C_DIS
LIN {X -0.084,Y -412.851,Z 527.505,A 0.000,B 0.000,C 90.000,E1 126.870} C_DIS
LIN {X -0.123,Y -412.853,Z 527.505,A 0.000,B 0.000,C 90.000,E1 126.870} C_DIS
LIN {X -0.069,Y -415.441,Z 527.500,A 0.000,B 0.000,C 90.000,E1 126.011} C_DIS
LIN {X -0.009,Y -425.839,Z 527.477,A 0.000,B 0.000,C 90.000,E1 121.926} C_DIS
LIN {X -0.066,Y -430.866,Z 527.468,A 0.000,B 0.000,C 90.000,E1 120.256} C_DIS
LIN {X -0.136,Y -439.910,Z 527.448,A 0.000,B 0.000,C 90.000,E1 116.616} C_DIS
LIN {X 0.050,Y -444.702,Z 527.439,A 0.000,B 0.000,C 90.000,E1 114.951} C_DIS
LIN {X 0.142,Y -451.427,Z 527.422,A 0.000,B 0.000,C 90.000,E1 111.972} C_DIS
LIN {X 0.106,Y -451.519,Z 527.422,A 0.000,B 0.000,C 90.000,E1 111.972} C_DIS
LIN {X 0.096,Y -476.500,Z 527.417,A 0.000,B 0.000,C 90.000,E1 111.046} C_DIS
LIN {X -0.108,Y -490.582,Z 527.414,A 0.000,B 0.000,C 90.000,E1 110.556} C_DIS
LIN {X 0.246,Y -500.816,Z 527.412,A 0.000,B 0.000,C 90.000,E1 110.120} C_DIS
LIN {X -0.176,Y -511.020,Z 527.410,A 0.000,B 0.000,C 90.000,E1 109.758} C_DIS
LIN {X 0.178,Y -524.722,Z 527.406,A 0.000,B 0.000,C 90.000,E1 109.141} C_DIS
LIN {X -0.113,Y -534.692,Z 527.404,A 0.000,B 0.000,C 90.000,E1 108.725} C_DIS
LIN {X -0.040,Y -544.525,Z 527.401,A 0.000,B 0.000,C 90.000,E1 108.236} C_DIS
LIN {X 0.100,Y -547.666,Z 527.400,A 0.000,B 0.000,C 90.000,E1 108.055} C_DIS
LIN {X -0.218,Y -552.315,Z 527.399,A 0.000,B 0.000,C 90.000,E1 107.819} C_DIS
LIN {X -0.150,Y -559.939,Z 527.396,A 0.000,B 0.000,C 90.000,E1 107.330} C_DIS
LIN {X 0.117,Y -565.333,Z 527.394,A 0.000,B 0.000,C 90.000,E1 106.913} C_DIS
LIN {X 0.144,Y -570.567,Z 527.392,A 0.000,B 0.000,C 90.000,E1 106.496} C_DIS
LIN {X 0.116,Y -574.716,Z 527.390,A 0.000,B 0.000,C 90.000,E1 106.150} C_DIS
LIN {X -0.073,Y -581.196,Z 527.386,A 0.000,B 0.000,C 90.000,E1 105.552} C_DIS
LIN {X 0.185,Y -586.213,Z 527.384,A 0.000,B 0.000,C 90.000,E1 105.009} C_DIS
LIN {X 0.038,Y -591.941,Z 527.380,A 0.000,B 0.000,C 90.000,E1 104.356} C_DIS
LIN {X 0.000,Y -596.291,Z 527.377,A 0.000,B 0.000,C 90.000,E1 103.828} C_DIS
LIN {X -0.292,Y -602.201,Z 527.372,A 0.000,B 0.000,C 90.000,E1 103.063} C_DIS
LIN {X 0.067,Y -607.819,Z 527.368,A 0.000,B 0.000,C 90.000,E1 102.243} C_DIS
LIN {X 0.259,Y -612.183,Z 527.365,A 0.000,B 0.000,C 90.000,E1 101.591} C_DIS
LIN {X -0.178,Y -614.805,Z 527.362,A 0.000,B 0.000,C 90.000,E1 101.243} C_DIS
LIN {X 0.199,Y -619.492,Z 527.358,A 0.000,B 0.000,C 90.000,E1 100.433} C_DIS
LIN {X 0.129,Y -623.814,Z 527.354,A 0.000,B 0.000,C 90.000,E1 99.670} C_DIS
LIN {X -0.186,Y -629.079,Z 527.348,A 0.000,B 0.000,C 90.000,E1 98.681} C_DIS
LIN {X 0.205,Y -633.400,Z 527.343,A 0.000,B 0.000,C 90.000,E1 97.757} C_DIS
LIN {X 0.324,Y -639.205,Z 527.336,A 0.000,B 0.000,C 90.000,E1 96.486} C_DIS
LIN {X 0.257,Y -642.583,Z 527.332,A 0.000,B 0.000,C 90.000,E1 95.739} C_DIS
LIN {X 0.227,Y -645.669,Z 527.328,A 0.000,B 0.000,C 90.000,E1 94.992} C_DIS
LIN {X 0.230,Y -648.541,Z 527.324,A 0.000,B 0.000,C 90.000,E1 94.245} C_DIS
LIN {X 0.262,Y -651.053,Z 527.320,A 0.000,B 0.000,C 90.000,E1 93.498} C_DIS
LIN {X 0.314,Y -653.270,Z 527.315,A 0.000,B 0.000,C 90.000,E1 92.751} C_DIS
LIN {X -0.295,Y -655.111,Z 527.311,A 0.000,B 0.000,C 90.000,E1 92.064} C_DIS
LIN {X -0.015,Y -656.124,Z 527.309,A 0.000,B 0.000,C 90.000,E1 91.547} C_DIS
LIN {X 0.252,Y -656.956,Z 527.306,A 0.000,B 0.000,C 90.000,E1 91.031} C_DIS
LIN {X -0.130,Y -657.595,Z 527.303,A 0.000,B 0.000,C 90.000,E1 90.573} C_DIS
LIN {X -0.037,Y -658.135,Z 527.299,A 0.000,B 0.000,C 90.000,E1 89.828} C_DIS
LIN {X 0.248,Y -658.321,Z 527.296,A 0.000,B 0.000,C 90.000,E1 89.312} C_DIS
LIN {X -0.124,Y -658.328,Z 527.294,A 0.000,B 0.000,C 90.000,E1 88.854} C_DIS
LIN {X 0.159,Y -658.160,Z 527.291,A 0.000,B 0.000,C 90.000,E1 88.339} C_DIS
LIN {X 0.275,Y -657.573,Z 527.287,A 0.000,B 0.000,C 90.000,E1 87.593} C_DIS
LIN {X -0.106,Y -657.027,Z 527.284,A 0.000,B 0.000,C 90.000,E1 87.135} C_DIS
LIN {X 0.004,Y -655.928,Z 527.280,A 0.000,B 0.000,C 90.000,E1 86.388} C_DIS
LIN {X -0.193,Y -655.516,Z 527.279,A 0.000,B 0.000,C 90.000,E1 86.159} C_DIS
LIN {X -0.096,Y -653.847,Z 527.275,A 0.000,B 0.000,C 90.000,E1 85.412} C_DIS
LIN {X 0.194,Y -652.647,Z 527.272,A 0.000,B 0.000,C 90.000,E1 84.894} C_DIS
LIN {X 0.108,Y -649.830,Z 527.266,A 0.000,B 0.000,C 90.000,E1 83.913} C_DIS
LIN {X 0.144,Y -647.331,Z 527.262,A 0.000,B 0.000,C 90.000,E1 83.166} C_DIS
LIN {X -0.250,Y -645.546,Z 527.259,A 0.000,B 0.000,C 90.000,E1 82.704} C_DIS
LIN {X -0.015,Y -643.628,Z 527.257,A 0.000,B 0.000,C 90.000,E1 82.186} C_DIS
LIN {X -0.132,Y -639.425,Z 527.251,A 0.000,B 0.000,C 90.000,E1 81.197} C_DIS
LIN {X -0.119,Y -635.897,Z 527.247,A 0.000,B 0.000,C 90.000,E1 80.443} C_DIS
LIN {X -0.184,Y -631.344,Z 527.242,A 0.000,B 0.000,C 90.000,E1 79.567} C_DIS
LIN {X -0.065,Y -628.617,Z 527.239,A 0.000,B 0.000,C 90.000,E1 79.050} C_DIS
LIN {X -0.260,Y -622.733,Z 527.234,A 0.000,B 0.000,C 90.000,E1 78.049} C_DIS
LIN {X -0.080,Y -619.634,Z 527.231,A 0.000,B 0.000,C 90.000,E1 77.521} C_DIS
LIN {X 0.079,Y -616.380,Z 527.228,A 0.000,B 0.000,C 90.000,E1 76.992} C_DIS
LIN {X 0.260,Y -613.713,Z 527.226,A 0.000,B 0.000,C 90.000,E1 76.589} C_DIS
LIN {X -0.273,Y -608.873,Z 527.222,A 0.000,B 0.000,C 90.000,E1 75.992} C_DIS
LIN {X 0.338,Y -603.372,Z 527.218,A 0.000,B 0.000,C 90.000,E1 75.283} C_DIS
LIN {X 0.334,Y -597.314,Z 527.215,A 0.000,B 0.000,C 90.000,E1 74.629} C_DIS
LIN {X -0.117,Y -593.501,Z 527.213,A 0.000,B 0.000,C 90.000,E1 74.283} C_DIS
LIN {X 0.292,Y -588.174,Z 527.210,A 0.000,B 0.000,C 90.000,E1 73.740} C_DIS
LIN {X 0.124,Y -582.430,Z 527.207,A 0.000,B 0.000,C 90.000,E1 73.268} C_DIS
LIN {X -0.200,Y -574.944,Z 527.204,A 0.000,B 0.000,C 90.000,E1 72.725} C_DIS
LIN {X -0.331,Y -568.741,Z 527.202,A 0.000,B 0.000,C 90.000,E1 72.308} C_DIS
LIN {X 0.130,Y -565.642,Z 527.200,A 0.000,B 0.000,C 90.000,E1 72.054} C_DIS
LIN {X 0.004,Y -559.154,Z 527.198,A 0.000,B 0.000,C 90.000,E1 71.692} C_DIS
LIN {X -0.230,Y -554.392,Z 527.197,A 0.000,B 0.000,C 90.000,E1 71.456} C_DIS
LIN {X -0.043,Y -545.687,Z 527.195,A 0.000,B 0.000,C 90.000,E1 71.040} C_DIS
LIN {X 0.265,Y -539.982,Z 527.193,A 0.000,B 0.000,C 90.000,E1 70.786} C_DIS
LIN {X 0.155,Y -536.874,Z 527.193,A 0.000,B 0.000,C 90.000,E1 70.678} C_DIS
LIN {X -0.164,Y -529.470,Z 527.191,A 0.000,B 0.000,C 90.000,E1 70.477} C_DIS
LIN {X 0.071,Y -518.306,Z 527.190,A 0.000,B 0.000,C 90.000,E1 70.134} C_DIS
LIN {X 0.193,Y -503.575,Z 527.188,A 0.000,B 0.000,C 90.000,E1 69.752} C_DIS
LIN {X 0.020,Y -492.400,Z 527.186,A 0.000,B 0.000,C 90.000,E1 69.518} C_DIS
LIN {X 0.118,Y -468.686,Z 527.184,A 0.000,B 0.000,C 90.000,E1 69.028} C_DIS
LIN {X 0.083,Y -468.558,Z 527.184,A 0.000,B 0.000,C 90.000,E1 69.028} C_DIS
LIN {X 0.159,Y -465.734,Z 527.173,A 0.000,B 0.000,C 90.000,E1 67.102} C_DIS
LIN {X -0.049,Y -461.555,Z 527.162,A 0.000,B 0.000,C 90.000,E1 65.229} C_DIS
LIN {X 0.059,Y -455.693,Z 527.145,A 0.000,B 0.000,C 90.000,E1 62.025} C_DIS
LIN {X -0.051,Y -455.028,Z 527.143,A 0.000,B 0.000,C 90.000,E1 61.719} C_DIS
LIN {X -0.154,Y -445.779,Z 527.120,A 0.000,B 0.000,C 90.000,E1 57.533} C_DIS
LIN {X -0.106,Y -445.030,Z 527.117,A 0.000,B 0.000,C 90.000,E1 57.120} C_DIS
LIN {X -0.145,Y -445.028,Z 527.117,A 0.000,B 0.000,C 90.000,E1 57.120} C_DIS
LIN {X 0.034,Y -448.210,Z 527.111,A 0.000,B 0.000,C 90.000,E1 55.881} C_DIS
LIN {X 0.129,Y -450.682,Z 527.105,A 0.000,B 0.000,C 90.000,E1 54.895} C_DIS
LIN {X -0.027,Y -453.639,Z 527.098,A 0.000,B 0.000,C 90.000,E1 53.623} C_DIS
LIN {X 0.132,Y -455.656,Z 527.093,A 0.000,B 0.000,C 90.000,E1 52.637} C_DIS
LIN {X -0.037,Y -458.023,Z 527.085,A 0.000,B 0.000,C 90.000,E1 51.376} C_DIS
LIN {X 0.189,Y -460.113,Z 527.078,A 0.000,B 0.000,C 90.000,E1 50.070} C_DIS
LIN {X -0.264,Y -461.963,Z 527.071,A 0.000,B 0.000,C 90.000,E1 48.852} C_DIS
LIN {X -0.088,Y -463.207,Z 527.066,A 0.000,B 0.000,C 90.000,E1 47.877} C_DIS
LIN {X 0.073,Y -464.248,Z 527.061,A 0.000,B 0.000,C 90.000,E1 46.905} C_DIS
LIN {X -0.068,Y -465.103,Z 527.055,A 0.000,B 0.000,C 90.000,E1 45.972} C_DIS
LIN {X 0.124,Y -465.802,Z 527.050,A 0.000,B 0.000,C 90.000,E1 45.000} C_DIS
LIN {X -0.012,Y -466.369,Z 527.045,A 0.000,B 0.000,C 90.000,E1 44.069} C_DIS
LIN {X -0.134,Y -466.739,Z 527.040,A 0.000,B 0.000,C 90.000,E1 43.137} C_DIS
LIN {X 0.163,Y -466.957,Z 527.033,A 0.000,B 0.000,C 90.000,E1 41.838} C_DIS
LIN {X 0.051,Y -466.981,Z 527.027,A 0.000,B 0.000,C 90.000,E1 40.906} C_DIS
LIN {X -0.010,Y -466.880,Z 527.022,A 0.000,B 0.000,C 90.000,E1 39.967} C_DIS
LIN {X 0.049,Y -466.475,Z 527.013,A 0.000,B 0.000,C 90.000,E1 38.382} C_DIS
LIN {X 0.164,Y -465.862,Z 527.005,A 0.000,B 0.000,C 90.000,E1 36.790} C_DIS
LIN {X -0.012,Y -465.112,Z 526.996,A 0.000,B 0.000,C 90.000,E1 35.231} C_DIS
LIN {X -0.082,Y -464.300,Z 526.987,A 0.000,B 0.000,C 90.000,E1 33.658} C_DIS
LIN {X 0.116,Y -463.076,Z 526.975,A 0.000,B 0.000,C 90.000,E1 31.416} C_DIS
LIN {X 0.263,Y -462.328,Z 526.968,A 0.000,B 0.000,C 90.000,E1 30.129} C_DIS
LIN {X 0.191,Y -461.126,Z 526.957,A 0.000,B 0.000,C 90.000,E1 28.231} C_DIS
LIN {X -0.123,Y -459.899,Z 526.946,A 0.000,B 0.000,C 90.000,E1 26.360} C_DIS
LIN {X -0.077,Y -459.185,Z 526.939,A 0.000,B 0.000,C 90.000,E1 25.079} C_DIS
LIN {X 0.007,Y -457.926,Z 526.925,A 0.000,B 0.000,C 90.000,E1 22.514} C_DIS
LIN {X 0.135,Y -456.947,Z 526.911,A 0.000,B 0.000,C 90.000,E1 19.939} C_DIS
LIN {X 0.172,Y -456.241,Z 526.898,A 0.000,B 0.000,C 90.000,E1 17.692} C_DIS
LIN {X -0.092,Y -455.846,Z 526.886,A 0.000,B 0.000,C 90.000,E1 15.481} C_DIS
LIN {X 0.165,Y -455.806,Z 526.872,A 0.000,B 0.000,C 90.000,E1 12.883} C_DIS
LIN {X 0.004,Y -456.129,Z 526.859,A 0.000,B 0.000,C 90.000,E1 10.658} C_DIS
LIN {X -0.087,Y -456.902,Z 526.845,A 0.000,B 0.000,C 90.000,E1 8.106} C_DIS
LIN {X 0.010,Y -457.898,Z 526.833,A 0.000,B 0.000,C 90.000,E1 5.853} C_DIS
LIN {X 0.044,Y -459.206,Z 526.820,A 0.000,B 0.000,C 90.000,E1 3.612} C_DIS
LIN {X 0.030,Y -461.393,Z 526.804,A 0.000,B 0.000,C 90.000,E1 0.745} C_DIS
LIN {X -0.172,Y -464.656,Z 526.787,A 0.000,B 0.000,C 90.000,E1 357.593} C_DIS
LIN {X -0.196,Y -466.922,Z 526.776,A 0.000,B 0.000,C 90.000,E1 355.698} C_DIS
LIN {X 0.091,Y -469.783,Z 526.764,A 0.000,B 0.000,C 90.000,E1 353.457} C_DIS
LIN {X 0.041,Y -471.948,Z 526.755,A 0.000,B 0.000,C 90.000,E1 351.894} C_DIS
LIN {X 0.036,Y -474.107,Z 526.746,A 0.000,B 0.000,C 90.000,E1 350.330} C_DIS
LIN {X -0.168,Y -477.261,Z 526.734,A 0.000,B 0.000,C 90.000,E1 348.173} C_DIS
LIN {X 0.092,Y -481.866,Z 526.719,A 0.000,B 0.000,C 90.000,E1 345.353} C_DIS
LIN {X -0.044,Y -486.661,Z 526.705,A 0.000,B 0.000,C 90.000,E1 342.906} C_DIS
LIN {X 0.212,Y -490.268,Z 526.695,A 0.000,B 0.000,C 90.000,E1 341.040} C_DIS
LIN {X -0.214,Y -494.005,Z 526.685,A 0.000,B 0.000,C 90.000,E1 339.263} C_DIS
LIN {X 0.090,Y -497.671,Z 526.675,A 0.000,B 0.000,C 90.000,E1 337.411} C_DIS
LIN {X -0.122,Y -500.007,Z 526.668,A 0.000,B 0.000,C 90.000,E1 336.230} C_DIS
LIN {X -0.023,Y -502.912,Z 526.660,A 0.000,B 0.000,C 90.000,E1 334.717} C_DIS
LIN {X 0.045,Y -505.175,Z 526.653,A 0.000,B 0.000,C 90.000,E1 333.512} C_DIS
LIN {X 0.090,Y -508.524,Z 526.643,A 0.000,B 0.000,C 90.000,E1 331.719} C_DIS
LIN {X -0.090,Y -511.309,Z 526.635,A 0.000,B 0.000,C 90.000,E1 330.255} C_DIS
LIN {X -0.213,Y -515.172,Z 526.623,A 0.000,B 0.000,C 90.000,E1 328.201} C_DIS
LIN {X 0.072,Y -517.492,Z 526.617,A 0.000,B 0.000,C 90.000,E1 326.993} C_DIS
LIN {X 0.186,Y -520.376,Z 526.609,A 0.000,B 0.000,C 90.000,E1 325.515} C_DIS
LIN {X 0.017,Y -523.786,Z 526.599,A 0.000,B 0.000,C 90.000,E1 323.783} C_DIS
LIN {X 0.090,Y -527.761,Z 526.588,A 0.000,B 0.000,C 90.000,E1 321.743} C_DIS
LIN {X -0.141,Y -531.726,Z 526.576,A 0.000,B 0.000,C 90.000,E1 319.747} C_DIS
LIN {X 0.074,Y -535.237,Z 526.567,A 0.000,B 0.000,C 90.000,E1 318.000} C_DIS
LIN {X -0.029,Y -538.274,Z 526.559,A 0.000,B 0.000,C 90.000,E1 316.581} C_DIS
LIN {X 0.298,Y -541.781,Z 526.549,A 0.000,B 0.000,C 90.000,E1 314.838} C_DIS
LIN {X -0.047,Y -546.604,Z 526.537,A 0.000,B 0.000,C 90.000,E1 312.609} C_DIS
LIN {X 0.136,Y -551.173,Z 526.526,A 0.000,B 0.000,C 90.000,E1 310.620} C_DIS
LIN {X 0.363,Y -554.271,Z 526.518,A 0.000,B 0.000,C 90.000,E1 309.197} C_DIS
LIN {X 0.218,Y -556.614,Z 526.512,A 0.000,B 0.000,C 90.000,E1 308.096} C_DIS
LIN {X 0.125,Y -561.106,Z 526.499,A 0.000,B 0.000,C 90.000,E1 305.884} C_DIS
LIN {X -0.368,Y -563.212,Z 526.495,A 0.000,B 0.000,C 90.000,E1 305.105} C_DIS
LIN {X -0.267,Y -564.118,Z 526.493,A 0.000,B 0.000,C 90.000,E1 304.818} C_DIS
LIN {X -0.271,Y -565.212,Z 526.491,A 0.000,B 0.000,C 90.000,E1 304.405} C_DIS
LIN {X 0.102,Y -566.490,Z 526.489,A 0.000,B 0.000,C 90.000,E1 304.040} C_DIS
LIN {X 0.110,Y -567.901,Z 526.487,A 0.000,B 0.000,C 90.000,E1 303.627} C_DIS
LIN {X -0.070,Y -570.125,Z 526.485,A 0.000,B 0.000,C 90.000,E1 303.245} C_DIS
LIN {X 0.230,Y -571.821,Z 526.483,A 0.000,B 0.000,C 90.000,E1 302.959} C_DIS
LIN {X 0.046,Y -573.365,Z 526.482,A 0.000,B 0.000,C 90.000,E1 302.704} C_DIS
LIN {X 0.179,Y -575.317,Z 526.480,A 0.000,B 0.000,C 90.000,E1 302.418} C_DIS
LIN {X 0.318,Y -576.801,Z 526.479,A 0.000,B 0.000,C 90.000,E1 302.133} C_DIS
LIN {X 0.312,Y -587.969,Z 526.470,A 0.000,B 0.000,C 90.000,E1 300.590} C_DIS
LIN {X 0.170,Y -591.134,Z 526.468,A 0.000,B 0.000,C 90.000,E1 300.207} C_DIS
LIN {X 0.113,Y -597.684,Z 526.463,A 0.000,B 0.000,C 90.000,E1 299.283} C_DIS
LIN {X -0.012,Y -600.274,Z 526.461,A 0.000,B 0.000,C 90.000,E1 298.899} C_DIS
LIN {X 0.066,Y -605.128,Z 526.456,A 0.000,B 0.000,C 90.000,E1 298.103} C_DIS
LIN {X 0.008,Y -606.592,Z 526.455,A 0.000,B 0.000,C 90.000,E1 297.847} C_DIS
LIN {X -0.116,Y -609.621,Z 526.451,A 0.000,B 0.000,C 90.000,E1 297.206} C_DIS
LIN {X 0.035,Y -611.790,Z 526.447,A 0.000,B 0.000,C 90.000,E1 296.411} C_DIS
LIN {X -0.001,Y -612.134,Z 526.445,A 0.000,B 0.000,C 90.000,E1 296.155} C_DIS
LIN {X -0.036,Y -612.280,Z 526.444,A 0.000,B 0.000,C 90.000,E1 295.899} C_DIS
LIN {X -0.070,Y -612.189,Z 526.443,A 0.000,B 0.000,C 90.000,E1 295.643} C_DIS
LIN {X 0.156,Y -611.463,Z 526.440,A 0.000,B 0.000,C 90.000,E1 295.103} C_DIS
LIN {X 0.123,Y -610.465,Z 526.438,A 0.000,B 0.000,C 90.000,E1 294.847} C_DIS
LIN {X 0.106,Y -609.814,Z 526.437,A 0.000,B 0.000,C 90.000,E1 294.719} C_DIS
LIN {X 0.088,Y -609.428,Z 526.437,A 0.000,B 0.000,C 90.000,E1 294.591} C_DIS
LIN {X 0.103,Y -608.641,Z 526.436,A 0.000,B 0.000,C 90.000,E1 294.387} C_DIS
LIN {X 0.058,Y -606.819,Z 526.434,A 0.000,B 0.000,C 90.000,E1 294.131} C_DIS
LIN {X 0.033,Y -605.752,Z 526.433,A 0.000,B 0.000,C 90.000,E1 294.003} C_DIS
LIN {X -0.224,Y -603.017,Z 526.432,A 0.000,B 0.000,C 90.000,E1 293.770} C_DIS
LIN {X -0.195,Y -596.724,Z 526.430,A 0.000,B 0.000,C 90.000,E1 293.334} C_DIS
LIN {X 0.014,Y -592.826,Z 526.429,A 0.000,B 0.000,C 90.000,E1 293.131} C_DIS
LIN {X 0.191,Y -584.021,Z 526.426,A 0.000,B 0.000,C 90.000,E1 292.589} C_DIS
LIN {X -0.103,Y -580.792,Z 526.424,A 0.000,B 0.000,C 90.000,E1 292.386} C_DIS
LIN {X -0.148,Y -579.532,Z 526.424,A 0.000,B 0.000,C 90.000,E1 292.280} C_DIS
LIN {X 0.027,Y -578.676,Z 526.423,A 0.000,B 0.000,C 90.000,E1 292.153} C_DIS
LIN {X 0.174,Y -578.205,Z 526.422,A 0.000,B 0.000,C 90.000,E1 292.025} C_DIS
LIN {X -0.055,Y -577.309,Z 526.420,A 0.000,B 0.000,C 90.000,E1 291.642} C_DIS
LIN {X 0.255,Y -577.330,Z 526.415,A 0.000,B 0.000,C 90.000,E1 290.663} C_DIS
LIN {X -0.254,Y -577.752,Z 526.409,A 0.000,B 0.000,C 90.000,E1 289.631} C_DIS
LIN {X 0.166,Y -577.864,Z 526.401,A 0.000,B 0.000,C 90.000,E1 288.236} C_DIS
LIN {X -0.142,Y -577.827,Z 526.394,A 0.000,B 0.000,C 90.000,E1 286.913} C_DIS
LIN {X -0.268,Y -577.602,Z 526.388,A 0.000,B 0.000,C 90.000,E1 285.843} C_DIS
LIN {X -0.180,Y -577.013,Z 526.377,A 0.000,B 0.000,C 90.000,E1 283.939} C_DIS
LIN {X -0.248,Y -576.542,Z 526.370,A 0.000,B 0.000,C 90.000,E1 282.591} C_DIS
LIN {X -0.109,Y -575.925,Z 526.361,A 0.000,B 0.000,C 90.000,E1 280.950} C_DIS
LIN {X 0.265,Y -575.373,Z 526.353,A 0.000,B 0.000,C 90.000,E1 279.557} C_DIS
LIN {X 0.181,Y -574.740,Z 526.344,A 0.000,B 0.000,C 90.000,E1 277.936} C_DIS
LIN {X -0.112,Y -574.300,Z 526.337,A 0.000,B 0.000,C 90.000,E1 276.606} C_DIS
LIN {X -0.288,Y -573.601,Z 526.328,A 0.000,B 0.000,C 90.000,E1 274.992} C_DIS
LIN {X -0.095,Y -572.897,Z 526.320,A 0.000,B 0.000,C 90.000,E1 273.612} C_DIS
LIN {X 0.048,Y -572.027,Z 526.313,A 0.000,B 0.000,C 90.000,E1 272.236} C_DIS
LIN {X -0.264,Y -570.814,Z 526.303,A 0.000,B 0.000,C 90.000,E1 270.630} C_DIS
LIN {X -0.042,Y -569.380,Z 526.294,A 0.000,B 0.000,C 90.000,E1 268.969} C_DIS
LIN {X 0.035,Y -568.175,Z 526.287,A 0.000,B 0.000,C 90.000,E1 267.593} C_DIS
LIN {X -0.024,Y -567.126,Z 526.281,A 0.000,B 0.000,C 90.000,E1 266.502} C_DIS
LIN {X 0.053,Y -565.892,Z 526.273,A 0.000,B 0.000,C 90.000,E1 265.122} C_DIS
LIN {X 0.106,Y -564.521,Z 526.265,A 0.000,B 0.000,C 90.000,E1 263.742} C_DIS
LIN {X 0.191,Y -562.971,Z 526.258,A 0.000,B 0.000,C 90.000,E1 262.356} C_DIS
LIN {X 0.243,Y -561.319,Z 526.250,A 0.000,B 0.000,C 90.000,E1 260.971} C_DIS
LIN {X 0.087,Y -558.875,Z 526.239,A 0.000,B 0.000,C 90.000,E1 259.050} C_DIS
LIN {X -0.155,Y -556.664,Z 526.230,A 0.000,B 0.000,C 90.000,E1 257.409} C_DIS
LIN {X 0.096,Y -554.542,Z 526.222,A 0.000,B 0.000,C 90.000,E1 255.992} C_DIS
LIN {X 0.191,Y -552.763,Z 526.216,A 0.000,B 0.000,C 90.000,E1 254.866} C_DIS
LIN {X 0.257,Y -550.793,Z 526.210,A 0.000,B 0.000,C 90.000,E1 253.740} C_DIS
LIN {X 0.190,Y -549.250,Z 526.205,A 0.000,B 0.000,C 90.000,E1 252.906} C_DIS
LIN {X 0.164,Y -545.772,Z 526.196,A 0.000,B 0.000,C 90.000,E1 251.221} C_DIS
LIN {X 0.210,Y -543.979,Z 526.191,A 0.000,B 0.000,C 90.000,E1 250.369} C_DIS
LIN {X 0.203,Y -540.825,Z 526.183,A 0.000,B 0.000,C 90.000,E1 248.954} C_DIS
LIN {X 0.194,Y -538.822,Z 526.179,A 0.000,B 0.000,C 90.000,E1 248.103} C_DIS
LIN {X 0.298,Y -535.355,Z 526.171,A 0.000,B 0.000,C 90.000,E1 246.666} C_DIS
LIN {X 0.143,Y -532.374,Z 526.164,A 0.000,B 0.000,C 90.000,E1 245.537} C_DIS
LIN {X 0.123,Y -528.491,Z 526.156,A 0.000,B 0.000,C 90.000,E1 244.101} C_DIS
LIN {X 0.089,Y -525.221,Z 526.150,A 0.000,B 0.000,C 90.000,E1 242.948} C_DIS
LIN {X 0.316,Y -520.319,Z 526.140,A 0.000,B 0.000,C 90.000,E1 241.179} C_DIS
LIN {X 0.073,Y -516.106,Z 526.132,A 0.000,B 0.000,C 90.000,E1 239.744} C_DIS
LIN {X -0.076,Y -512.639,Z 526.125,A 0.000,B 0.000,C 90.000,E1 238.584} C_DIS
LIN {X 0.123,Y -507.218,Z 526.116,A 0.000,B 0.000,C 90.000,E1 236.786} C_DIS
LIN {X 0.086,Y -499.860,Z 526.102,A 0.000,B 0.000,C 90.000,E1 234.402} C_DIS
LIN {X -0.117,Y -493.834,Z 526.091,A 0.000,B 0.000,C 90.000,E1 232.316} C_DIS
LIN {X -0.007,Y -490.445,Z 526.084,A 0.000,B 0.000,C 90.000,E1 231.090} C_DIS
LIN {X 0.184,Y -486.263,Z 526.075,A 0.000,B 0.000,C 90.000,E1 229.542} C_DIS
LIN {X 0.177,Y -480.604,Z 526.063,A 0.000,B 0.000,C 90.000,E1 227.391} C_DIS
LIN {X -0.006,Y -477.376,Z 526.057,A 0.000,B 0.000,C 90.000,E1 226.176} C_DIS
LIN {X 0.211,Y -473.524,Z 526.048,A 0.000,B 0.000,C 90.000,E1 224.595} C_DIS
LIN {X -0.076,Y -470.470,Z 526.041,A 0.000,B 0.000,C 90.000,E1 223.380} C_DIS
LIN {X -0.313,Y -466.739,Z 526.032,A 0.000,B 0.000,C 90.000,E1 221.838} C_DIS
LIN {X 0.035,Y -463.171,Z 526.023,A 0.000,B 0.000,C 90.000,E1 220.216} C_DIS
LIN {X -0.163,Y -458.194,Z 526.011,A 0.000,B 0.000,C 90.000,E1 218.016} C_DIS
LIN {X 0.148,Y -454.738,Z 526.002,A 0.000,B 0.000,C 90.000,E1 216.377} C_DIS
LIN {X 0.181,Y -450.040,Z 525.990,A 0.000,B 0.000,C 90.000,E1 214.119} C_DIS
LIN {X -0.041,Y -445.585,Z 525.977,A 0.000,B 0.000,C 90.000,E1 211.878} C_DIS
LIN {X -0.008,Y -441.261,Z 525.964,A 0.000,B 0.000,C 90.000,E1 209.589} C_DIS
LIN {X -0.184,Y -437.810,Z 525.953,A 0.000,B 0.000,C 90.000,E1 207.641} C_DIS
LIN {X -0.056,Y -434.404,Z 525.942,A 0.000,B 0.000,C 90.000,E1 205.643} C_DIS
LIN {X 0.206,Y -430.005,Z 525.928,A 0.000,B 0.000,C 90.000,E1 202.950} C_DIS
LIN {X 0.004,Y -426.003,Z 525.913,A 0.000,B 0.000,C 90.000,E1 200.301} C_DIS
LIN {X -0.046,Y -423.221,Z 525.902,A 0.000,B 0.000,C 90.000,E1 198.290} C_DIS
LIN {X 0.150,Y -420.273,Z 525.888,A 0.000,B 0.000,C 90.000,E1 195.898} C_DIS
LIN {X -0.008,Y -417.822,Z 525.877,A 0.000,B 0.000,C 90.000,E1 193.883} C_DIS
LIN {X -0.181,Y -414.213,Z 525.860,A 0.000,B 0.000,C 90.000,E1 190.838} C_DIS
LIN {X 0.038,Y -412.382,Z 525.851,A 0.000,B 0.000,C 90.000,E1 189.095} C_DIS
LIN {X 0.184,Y -410.955,Z 525.843,A 0.000,B 0.000,C 90.000,E1 187.701} C_DIS
LIN {X -0.144,Y -408.392,Z 525.830,A 0.000,B 0.000,C 90.000,E1 185.334} C_DIS
LIN {X 0.106,Y -405.140,Z 525.808,A 0.000,B 0.000,C 90.000,E1 181.489} C_DIS
LIN {X -0.093,Y -403.532,Z 525.795,A 0.000,B 0.000,C 90.000,E1 179.083} C_DIS
LIN {X 0.038,Y -402.154,Z 525.777,A 0.000,B 0.000,C 90.000,E1 175.927} C_DIS
LIN {X 0.186,Y -401.469,Z 525.760,A 0.000,B 0.000,C 90.000,E1 172.761} C_DIS
LIN {X 0.080,Y -401.359,Z 525.748,A 0.000,B 0.000,C 90.000,E1 170.679} C_DIS
LIN {X 0.096,Y -401.526,Z 525.735,A 0.000,B 0.000,C 90.000,E1 168.229} C_DIS
LIN {X -0.025,Y -402.243,Z 525.717,A 0.000,B 0.000,C 90.000,E1 165.102} C_DIS
LIN {X -0.008,Y -403.283,Z 525.702,A 0.000,B 0.000,C 90.000,E1 162.308} C_DIS
LIN {X 0.000,Y -403.969,Z 525.694,A 0.000,B 0.000,C 90.000,E1 160.913} C_DIS
LIN {X -0.084,Y -405.824,Z 525.677,A 0.000,B 0.000,C 90.000,E1 157.794} C_DIS
LIN {X -0.018,Y -407.983,Z 525.659,A 0.000,B 0.000,C 90.000,E1 154.665} C_DIS
LIN {X -0.189,Y -409.514,Z 525.648,A 0.000,B 0.000,C 90.000,E1 152.615} C_DIS
LIN {X -0.139,Y -410.965,Z 525.636,A 0.000,B 0.000,C 90.000,E1 150.539} C_DIS
LIN {X 0.134,Y -411.806,Z 525.629,A 0.000,B 0.000,C 90.000,E1 149.125} C_DIS
LIN {X -0.206,Y -412.732,Z 525.619,A 0.000,B 0.000,C 90.000,E1 147.454} C_DIS
LIN {X -0.182,Y -413.262,Z 525.613,A 0.000,B 0.000,C 90.000,E1 146.421} C_DIS
LIN {X 0.123,Y -414.167,Z 525.602,A 0.000,B 0.000,C 90.000,E1 144.322} C_DIS
LIN {X -0.175,Y -414.561,Z 525.596,A 0.000,B 0.000,C 90.000,E1 143.336} C_DIS
LIN {X -0.114,Y -415.106,Z 525.587,A 0.000,B 0.000,C 90.000,E1 141.618} C_DIS
LIN {X -0.113,Y -415.578,Z 525.577,A 0.000,B 0.000,C 90.000,E1 139.908} C_DIS
LIN {X 0.168,Y -415.964,Z 525.568,A 0.000,B 0.000,C 90.000,E1 138.162} C_DIS
LIN {X 0.017,Y -416.162,Z 525.556,A 0.000,B 0.000,C 90.000,E1 136.134} C_DIS
LIN {X 0.108,Y -416.214,Z 525.549,A 0.000,B 0.000,C 90.000,E1 134.757} C_DIS
LIN {X -0.089,Y -416.153,Z 525.541,A 0.000,B 0.000,C 90.000,E1 133.419} C_DIS
LIN {X 0.121,Y -416.029,Z 525.536,A 0.000,B 0.000,C 90.000,E1 132.366} C_DIS
LIN {X 0.042,Y -415.755,Z 525.530,A 0.000,B 0.000,C 90.000,E1 131.353} C_DIS
LIN {X 0.002,Y -415.340,Z 525.524,A 0.000,B 0.000,C 90.000,E1 130.334} C_DIS
LIN {X 0.088,Y -414.538,Z 525.517,A 0.000,B 0.000,C 90.000,E1 128.955} C_DIS
LIN {X 0.136,Y -413.419,Z 525.507,A 0.000,B 0.000,C 90.000,E1 127.237} C_DIS
LIN {X -0.115,Y -413.105,Z 525.504,A 0.000,B 0.000,C 90.000,E1 126.790} C_DIS
LIN {X -0.154,Y -413.104,Z 525.504,A 0.000,B 0.000,C 90.000,E1 126.790} C_DIS
LIN {X 0.003,Y -415.759,Z 525.499,A 0.000,B 0.000,C 90.000,E1 125.884} C_DIS
LIN {X 0.110,Y -425.205,Z 525.479,A 0.000,B 0.000,C 90.000,E1 122.133} C_DIS
LIN {X 0.043,Y -430.204,Z 525.469,A 0.000,B 0.000,C 90.000,E1 120.463} C_DIS
LIN {X 0.042,Y -431.120,Z 525.467,A 0.000,B 0.000,C 90.000,E1 120.129} C_DIS
LIN {X -0.011,Y -440.222,Z 525.447,A 0.000,B 0.000,C 90.000,E1 116.488} C_DIS
LIN {X -0.005,Y -444.973,Z 525.438,A 0.000,B 0.000,C 90.000,E1 114.847} C_DIS
LIN {X 0.083,Y -452.223,Z 525.420,A 0.000,B 0.000,C 90.000,E1 111.663} C_DIS
LIN {X 0.043,Y -452.245,Z 525.420,A 0.000,B 0.000,C 90.000,E1 111.663} C_DIS
LIN {X -0.271,Y -478.781,Z 525.415,A 0.000,B 0.000,C 90.000,E1 110.737} C_DIS
LIN {X 0.204,Y -492.823,Z 525.412,A 0.000,B 0.000,C 90.000,E1 110.174} C_DIS
LIN {X 0.004,Y -499.679,Z 525.411,A 0.000,B 0.000,C 90.000,E1 109.939} C_DIS
LIN {X -0.038,Y -513.367,Z 525.408,A 0.000,B 0.000,C 90.000,E1 109.396} C_DIS
LIN {X 0.021,Y -523.694,Z 525.405,A 0.000,B 0.000,C 90.000,E1 108.960} C_DIS
LIN {X -0.209,Y -533.853,Z 525.403,A 0.000,B 0.000,C 90.000,E1 108.544} C_DIS
LIN {X -0.203,Y -540.429,Z 525.401,A 0.000,B 0.000,C 90.000,E1 108.236} C_DIS
LIN {X 0.212,Y -546.783,Z 525.399,A 0.000,B 0.000,C 90.000,E1 107.873} C_DIS
LIN {X 0.184,Y -555.954,Z 525.397,A 0.000,B 0.000,C 90.000,E1 107.347} C_DIS
LIN {X -0.120,Y -560.372,Z 525.395,A 0.000,B 0.000,C 90.000,E1 107.094} C_DIS
LIN {X 0.140,Y -565.869,Z 525.393,A 0.000,B 0.000,C 90.000,E1 106.677} C_DIS
LIN {X -0.214,Y -568.832,Z 525.392,A 0.000,B 0.000,C 90.000,E1 106.496} C_DIS
LIN {X -0.113,Y -574.435,Z 525.389,A 0.000,B 0.000,C 90.000,E1 106.024} C_DIS
LIN {X -0.110,Y -579.788,Z 525.386,A 0.000,B 0.000,C 90.000,E1 105.536} C_DIS
LIN {X -0.106,Y -586.104,Z 525.383,A 0.000,B 0.000,C 90.000,E1 104.898} C_DIS
LIN {X -0.021,Y -590.884,Z 525.380,A 0.000,B 0.000,C 90.000,E1 104.356} C_DIS
LIN {X -0.127,Y -596.392,Z 525.376,A 0.000,B 0.000,C 90.000,E1 103.703} C_DIS
LIN {X -0.031,Y -602.174,Z 525.372,A 0.000,B 0.000,C 90.000,E1 102.939} C_DIS
LIN {X 0.240,Y -605.951,Z 525.369,A 0.000,B 0.000,C 90.000,E1 102.411} C_DIS
LIN {X 0.106,Y -610.642,Z 525.365,A 0.000,B 0.000,C 90.000,E1 101.771} C_DIS
LIN {X 0.221,Y -615.714,Z 525.361,A 0.000,B 0.000,C 90.000,E1 101.007} C_DIS
LIN {X 0.259,Y -620.343,Z 525.357,A 0.000,B 0.000,C 90.000,E1 100.254} C_DIS
LIN {X 0.089,Y -624.760,Z 525.353,A 0.000,B 0.000,C 90.000,E1 99.500} C_DIS
LIN {X -0.092,Y -629.462,Z 525.348,A 0.000,B 0.000,C 90.000,E1 98.624} C_DIS
LIN {X 0.165,Y -634.462,Z 525.342,A 0.000,B 0.000,C 90.000,E1 97.587} C_DIS
LIN {X -0.005,Y -638.582,Z 525.337,A 0.000,B 0.000,C 90.000,E1 96.720} C_DIS
LIN {X -0.262,Y -643.144,Z 525.332,A 0.000,B 0.000,C 90.000,E1 95.739} C_DIS
LIN {X -0.289,Y -646.263,Z 525.328,A 0.000,B 0.000,C 90.000,E1 94.992} C_DIS
LIN {X -0.055,Y -648.219,Z 525.325,A 0.000,B 0.000,C 90.000,E1 94.473} C_DIS
LIN {X -0.031,Y -650.837,Z 525.321,A 0.000,B 0.000,C 90.000,E1 93.726} C_DIS
LIN {X 0.193,Y -652.448,Z 525.318,A 0.000,B 0.000,C 90.000,E1 93.212} C_DIS
LIN {X -0.189,Y -653.889,Z 525.315,A 0.000,B 0.000,C 90.000,E1 92.751} C_DIS
LIN {X -0.139,Y -655.745,Z 525.311,A 0.000,B 0.000,C 90.000,E1 92.007} C_DIS
LIN {X -0.048,Y -657.204,Z 525.307,A 0.000,B 0.000,C 90.000,E1 91.260} C_DIS
LIN {X 0.040,Y -658.168,Z 525.303,A 0.000,B 0.000,C 90.000,E1 90.516} C_DIS
LIN {X 0.139,Y -658.672,Z 525.299,A 0.000,B 0.000,C 90.000,E1 89.771} C_DIS
LIN {X -0.047,Y -658.810,Z 525.297,A 0.000,B 0.000,C 90.000,E1 89.542} C_DIS
LIN {X 0.057,Y -658.805,Z 525.293,A 0.000,B 0.000,C 90.000,E1 88.797} C_DIS
LIN {X -0.314,Y -658.595,Z 525.291,A 0.000,B 0.000,C 90.000,E1 88.339} C_DIS
LIN {X -0.194,Y -657.972,Z 525.287,A 0.000,B 0.000,C 90.000,E1 87.593} C_DIS
LIN {X 0.275,Y -657.743,Z 525.285,A 0.000,B 0.000,C 90.000,E1 87.306} C_DIS
LIN {X -0.263,Y -656.630,Z 525.281,A 0.000,B 0.000,C 90.000,E1 86.617} C_DIS
LIN {X 0.001,Y -655.780,Z 525.278,A 0.000,B 0.000,C 90.000,E1 86.102} C_DIS
LIN {X 0.099,Y -654.075,Z 525.274,A 0.000,B 0.000,C 90.000,E1 85.355} C_DIS
LIN {X -0.259,Y -652.804,Z 525.272,A 0.000,B 0.000,C 90.000,E1 84.894} C_DIS
LIN {X 0.305,Y -649.880,Z 525.266,A 0.000,B 0.000,C 90.000,E1 83.856} C_DIS
LIN {X -0.302,Y -647.285,Z 525.262,A 0.000,B 0.000,C 90.000,E1 83.166} C_DIS
LIN {X -0.214,Y -644.389,Z 525.258,A 0.000,B 0.000,C 90.000,E1 82.413} C_DIS
LIN {X 0.014,Y -642.320,Z 525.255,A 0.000,B 0.000,C 90.000,E1 81.894} C_DIS
LIN {X 0.224,Y -640.184,Z 525.252,A 0.000,B 0.000,C 90.000,E1 81.376} C_DIS
LIN {X 0.203,Y -635.991,Z 525.247,A 0.000,B 0.000,C 90.000,E1 80.500} C_DIS
LIN {X -0.264,Y -633.381,Z 525.245,A 0.000,B 0.000,C 90.000,E1 80.038} C_DIS
LIN {X -0.206,Y -629.276,Z 525.240,A 0.000,B 0.000,C 90.000,E1 79.275} C_DIS
LIN {X 0.313,Y -623.381,Z 525.235,A 0.000,B 0.000,C 90.000,E1 78.229} C_DIS
LIN {X 0.273,Y -618.627,Z 525.231,A 0.000,B 0.000,C 90.000,E1 77.465} C_DIS
LIN {X 0.186,Y -613.382,Z 525.226,A 0.000,B 0.000,C 90.000,E1 76.700} C_DIS
LIN {X 0.099,Y -608.443,Z 525.223,A 0.000,B 0.000,C 90.000,E1 76.061} C_DIS
LIN {X 0.202,Y -602.894,Z 525.219,A 0.000,B 0.000,C 90.000,E1 75.408} C_DIS
LIN {X 0.227,Y -596.711,Z 525.215,A 0.000,B 0.000,C 90.000,E1 74.755} C_DIS
LIN {X 0.016,Y -592.915,Z 525.213,A 0.000,B 0.000,C 90.000,E1 74.393} C_DIS
LIN {X -0.210,Y -587.527,Z 525.211,A 0.000,B 0.000,C 90.000,E1 73.921} C_DIS
LIN {X -0.034,Y -581.851,Z 525.208,A 0.000,B 0.000,C 90.000,E1 73.433} C_DIS
LIN {X 0.194,Y -575.938,Z 525.206,A 0.000,B 0.000,C 90.000,E1 72.960} C_DIS
LIN {X 0.087,Y -569.784,Z 525.203,A 0.000,B 0.000,C 90.000,E1 72.543} C_DIS
LIN {X 0.081,Y -565.042,Z 525.201,A 0.000,B 0.000,C 90.000,E1 72.236} C_DIS
LIN {X -0.139,Y -558.174,Z 525.199,A 0.000,B 0.000,C 90.000,E1 71.873} C_DIS
LIN {X 0.144,Y -553.170,Z 525.198,A 0.000,B 0.000,C 90.000,E1 71.583} C_DIS
LIN {X 0.186,Y -546.284,Z 525.196,A 0.000,B 0.000,C 90.000,E1 71.275} C_DIS
LIN {X -0.160,Y -539.131,Z 525.195,A 0.000,B 0.000,C 90.000,E1 71.040} C_DIS
LIN {X -0.147,Y -535.741,Z 525.194,A 0.000,B 0.000,C 90.000,E1 70.913} C_DIS
LIN {X 0.292,Y -526.770,Z 525.192,A 0.000,B 0.000,C 90.000,E1 70.604} C_DIS
LIN {X -0.286,Y -515.783,Z 525.191,A 0.000,B 0.000,C 90.000,E1 70.369} C_DIS
LIN {X -0.254,Y -502.940,Z 525.189,A 0.000,B 0.000,C 90.000,E1 70.061} C_DIS
LIN {X 0.041,Y -493.438,Z 525.188,A 0.000,B 0.000,C 90.000,E1 69.826} C_DIS
LIN {X 0.143,Y -471.376,Z 525.186,A 0.000,B 0.000,C 90.000,E1 69.390} C_DIS
LIN {X -0.178,Y -469.237,Z 525.185,A 0.000,B 0.000,C 90.000,E1 69.390} C_DIS
LIN {X -0.214,Y -469.095,Z 525.185,A 0.000,B 0.000,C 90.000,E1 69.390} C_DIS
LIN {X 0.253,Y -465.750,Z 525.173,A 0.000,B 0.000,C 90.000,E1 67.102} C_DIS
LIN {X 0.068,Y -463.643,Z 525.168,A 0.000,B 0.000,C 90.000,E1 66.177} C_DIS
LIN {X 0.153,Y -455.711,Z 525.145,A 0.000,B 0.000,C 90.000,E1 62.025} C_DIS
LIN {X 0.043,Y -455.058,Z 525.143,A 0.000,B 0.000,C 90.000,E1 61.719} C_DIS
LIN {X -0.130,Y -446.418,Z 525.121,A 0.000,B 0.000,C 90.000,E1 57.867} C_DIS
LIN {X -0.072,Y -445.358,Z 525.118,A 0.000,B 0.000,C 90.000,E1 57.296} C_DIS
LIN {X 0.262,Y -445.363,Z 525.118,A 0.000,B 0.000,C 90.000,E1 57.248} C_DIS
LIN {X 0.135,Y -449.151,Z 525.111,A 0.000,B 0.000,C 90.000,E1 55.881} C_DIS
LIN {X 0.242,Y -451.640,Z 525.105,A 0.000,B 0.000,C 90.000,E1 54.895} C_DIS
LIN {X 0.100,Y -454.659,Z 525.098,A 0.000,B 0.000,C 90.000,E1 53.623} C_DIS
LIN {X -0.091,Y -456.712,Z 525.093,A 0.000,B 0.000,C 90.000,E1 52.683} C_DIS
LIN {X 0.102,Y -458.512,Z 525.087,A 0.000,B 0.000,C 90.000,E1 51.698} C_DIS
LIN {X -0.024,Y -460.600,Z 525.080,A 0.000,B 0.000,C 90.000,E1 50.436} C_DIS
LIN {X -0.120,Y -462.498,Z 525.073,A 0.000,B 0.000,C 90.000,E1 49.175} C_DIS
LIN {X 0.113,Y -464.114,Z 525.066,A 0.000,B 0.000,C 90.000,E1 47.877} C_DIS
LIN {X -0.032,Y -465.131,Z 525.061,A 0.000,B 0.000,C 90.000,E1 46.944} C_DIS
LIN {X 0.155,Y -465.960,Z 525.056,A 0.000,B 0.000,C 90.000,E1 45.972} C_DIS
LIN {X 0.027,Y -466.640,Z 525.050,A 0.000,B 0.000,C 90.000,E1 45.040} C_DIS
LIN {X -0.094,Y -467.203,Z 525.045,A 0.000,B 0.000,C 90.000,E1 44.109} C_DIS
LIN {X -0.129,Y -467.621,Z 525.038,A 0.000,B 0.000,C 90.000,E1 42.852} C_DIS
LIN {X -0.161,Y -467.810,Z 525.031,A 0.000,B 0.000,C 90.000,E1 41.595} C_DIS
LIN {X -0.084,Y -467.654,Z 525.022,A 0.000,B 0.000,C 90.000,E1 40.011} C_DIS
LIN {X 0.057,Y -467.218,Z 525.014,A 0.000,B 0.000,C 90.000,E1 38.418} C_DIS
LIN {X -0.176,Y -466.606,Z 525.005,A 0.000,B 0.000,C 90.000,E1 36.870} C_DIS
LIN {X 0.046,Y -465.830,Z 524.996,A 0.000,B 0.000,C 90.000,E1 35.264} C_DIS
LIN {X -0.130,Y -465.005,Z 524.987,A 0.000,B 0.000,C 90.000,E1 33.706} C_DIS
LIN {X 0.078,Y -463.734,Z 524.975,A 0.000,B 0.000,C 90.000,E1 31.465} C_DIS
LIN {X -0.003,Y -462.958,Z 524.968,A 0.000,B 0.000,C 90.000,E1 30.207} C_DIS
LIN {X 0.036,Y -461.924,Z 524.959,A 0.000,B 0.000,C 90.000,E1 28.615} C_DIS
LIN {X -0.261,Y -460.656,Z 524.948,A 0.000,B 0.000,C 90.000,E1 26.744} C_DIS
LIN {X -0.289,Y -459.713,Z 524.940,A 0.000,B 0.000,C 90.000,E1 25.155} C_DIS
LIN {X -0.092,Y -458.561,Z 524.927,A 0.000,B 0.000,C 90.000,E1 22.898} C_DIS
LIN {X -0.112,Y -457.597,Z 524.915,A 0.000,B 0.000,C 90.000,E1 20.663} C_DIS
LIN {X -0.207,Y -457.162,Z 524.908,A 0.000,B 0.000,C 90.000,E1 19.396} C_DIS
LIN {X -0.165,Y -456.461,Z 524.895,A 0.000,B 0.000,C 90.000,E1 17.149} C_DIS
LIN {X 0.223,Y -456.114,Z 524.881,A 0.000,B 0.000,C 90.000,E1 14.537} C_DIS
LIN {X -0.056,Y -456.206,Z 524.867,A 0.000,B 0.000,C 90.000,E1 12.007} C_DIS
LIN {X -0.061,Y -456.696,Z 524.852,A 0.000,B 0.000,C 90.000,E1 9.443} C_DIS
LIN {X -0.130,Y -457.622,Z 524.838,A 0.000,B 0.000,C 90.000,E1 6.891} C_DIS
LIN {X 0.119,Y -458.964,Z 524.824,A 0.000,B 0.000,C 90.000,E1 4.302} C_DIS
LIN {X 0.160,Y -460.459,Z 524.812,A 0.000,B 0.000,C 90.000,E1 2.064} C_DIS
END
